LIN {X 0,Y 441.31,Z 713.297,A -85,B 0,C 180,E1 21599.481,E2 21599.481} C_VEL
LIN {X 0,Y 441.247,Z 716.806,A -85,B 0,C 180,E1 21597.403,E2 21597.403} C_VEL
LIN {X 0,Y 441.266,Z 718.402,A -85,B 0,C 180,E1 21595.322,E2 21595.322} C_VEL
LIN {X 0,Y 441.352,Z 718.291,A -85,B 0,C 180,E1 21593.366,E2 21593.366} C_VEL
LIN {X 0,Y 441.5,Z 716.286,A -85,B 0,C 180,E1 21591.273,E2 21591.273} C_VEL
LIN {X 0,Y 441.746,Z 712.662,A -85,B 0,C 180,E1 21589.304,E2 21589.304} C_VEL
LIN {X 0,Y 442.049,Z 707.079,A -85,B 0,C 180,E1 21587.327,E2 21587.327} C_VEL
LIN {X 0,Y 442.464,Z 699.897,A -85,B 0,C 180,E1 21585.474,E2 21585.474} C_VEL
LIN {X 0,Y 442.948,Z 691.121,A -85,B 0,C 180,E1 21583.746,E2 21583.746} C_VEL
LIN {X 0,Y 443.459,Z 681.227,A -85,B 0,C 180,E1 21582.212,E2 21582.212} C_VEL
LIN {X 0,Y 444.021,Z 669.276,A -85,B 0,C 180,E1 21580.738,E2 21580.738} C_VEL
LIN {X 0,Y 444.497,Z 656.854,A -85,B 0,C 180,E1 21579.526,E2 21579.526} C_VEL
LIN {X 0,Y 444.916,Z 642.754,A -85,B 0,C 180,E1 21578.443,E2 21578.443} C_VEL
LIN {X 0,Y 445.197,Z 627.324,A -85,B 0,C 180,E1 21577.555,E2 21577.555} C_VEL
LIN {X 0,Y 445.338,Z 611.674,A -85,B 0,C 180,E1 21576.911,E2 21576.911} C_VEL
LIN {X 0,Y 445.29,Z 594.343,A -85,B 0,C 180,E1 21576.46,E2 21576.46} C_VEL
LIN {X 0,Y 446.556,Z 505.792,A -85,B 0,C 180,E1 21574.804,E2 21574.804} C_VEL
LIN {X 0,Y 447.572,Z 462.908,A -85,B 0,C 180,E1 21573.926,E2 21573.926} C_VEL
LIN {X 0,Y 449.09,Z 454.637,A -85,B 0,C 180,E1 21573.345,E2 21573.345} C_VEL
LIN {X 0,Y 449.865,Z 411.959,A -85,B 0,C 180,E1 21569.922,E2 21569.922} C_VEL
LIN {X 0,Y 450.238,Z 377.811,A -85,B 0,C 180,E1 21567.266,E2 21567.266} C_VEL
LIN {X 0,Y 450.427,Z 358.214,A -85,B 0,C 180,E1 21565.756,E2 21565.756} C_VEL
LIN {X 0,Y 452.726,Z 358.689,A -85,B 0,C 180,E1 21565.418,E2 21565.418} C_VEL
LIN {X 0,Y 455.691,Z 357.568,A -85,B 0,C 180,E1 21565.147,E2 21565.147} C_VEL
LIN {X 0,Y 456.996,Z 357.12,A -85,B 0,C 180,E1 21565.025,E2 21565.025} C_VEL
LIN {X 0,Y 461.236,Z 356.094,A -85,B 0,C 180,E1 21564.597,E2 21564.597} C_VEL
LIN {X 0,Y 470.221,Z 353.87,A -85,B 0,C 180,E1 21563.727,E2 21563.727} C_VEL
LIN {X 0,Y 470.656,Z 372.168,A -85,B 0,C 180,E1 21562.125,E2 21562.125} C_VEL
LIN {X 0,Y 472.911,Z 388.879,A -85,B 0,C 180,E1 21560.508,E2 21560.508} C_VEL
LIN {X 0,Y 476.938,Z 403.833,A -85,B 0,C 180,E1 21558.912,E2 21558.912} C_VEL
LIN {X 0,Y 482.198,Z 416.087,A -85,B 0,C 180,E1 21557.471,E2 21557.471} C_VEL
LIN {X 0,Y 489.251,Z 427.616,A -85,B 0,C 180,E1 21555.986,E2 21555.986} C_VEL
LIN {X 0,Y 498.516,Z 438.468,A -85,B 0,C 180,E1 21554.438,E2 21554.438} C_VEL
LIN {X 0,Y 508.804,Z 447.18,A -85,B 0,C 180,E1 21553.028,E2 21553.028} C_VEL
LIN {X 0,Y 517.76,Z 453.161,A -85,B 0,C 180,E1 21551.96,E2 21551.96} C_VEL
LIN {X 0,Y 501.787,Z 477.95,A -85,B 0,C 180,E1 21551.418,E2 21551.418} C_VEL
LIN {X 0,Y 491.807,Z 495.847,A -85,B 0,C 180,E1 21550.892,E2 21550.892} C_VEL
LIN {X 0,Y 483.679,Z 513.365,A -85,B 0,C 180,E1 21550.241,E2 21550.241} C_VEL
LIN {X 0,Y 476.055,Z 528.839,A -85,B 0,C 180,E1 21549.68,E2 21549.68} C_VEL
LIN {X 0,Y 467.291,Z 551.983,A -85,B 0,C 180,E1 21548.665,E2 21548.665} C_VEL
LIN {X 0,Y 465.606,Z 571.959,A -85,B 0,C 180,E1 21548.437,E2 21548.437} C_VEL
LIN {X 0,Y 464.664,Z 601.449,A -85,B 0,C 180,E1 21547.884,E2 21547.884} C_VEL
LIN {X 0,Y 462.976,Z 626.356,A -85,B 0,C 180,E1 21547.202,E2 21547.202} C_VEL
LIN {X 0,Y 461.15,Z 649.493,A -85,B 0,C 180,E1 21546.332,E2 21546.332} C_VEL
LIN {X 0,Y 459.06,Z 672.171,A -85,B 0,C 180,E1 21545.238,E2 21545.238} C_VEL
LIN {X 0,Y 456.925,Z 693.284,A -85,B 0,C 180,E1 21543.969,E2 21543.969} C_VEL
LIN {X 0,Y 454.675,Z 713.158,A -85,B 0,C 180,E1 21542.525,E2 21542.525} C_VEL
LIN {X 0,Y 452.365,Z 732.465,A -85,B 0,C 180,E1 21540.85,E2 21540.85} C_VEL
LIN {X 0,Y 450.053,Z 750.796,A -85,B 0,C 180,E1 21538.968,E2 21538.968} C_VEL
LIN {X 0,Y 448.043,Z 766.471,A -85,B 0,C 180,E1 21537.076,E2 21537.076} C_VEL
LIN {X 0,Y 445.95,Z 782.819,A -85,B 0,C 180,E1 21534.764,E2 21534.764} C_VEL
LIN {X 0,Y 444.103,Z 797.993,A -85,B 0,C 180,E1 21532.225,E2 21532.225} C_VEL
LIN {X 0,Y 442.674,Z 810.867,A -85,B 0,C 180,E1 21529.667,E2 21529.667} C_VEL
LIN {X 0,Y 441.61,Z 821.723,A -85,B 0,C 180,E1 21527.118,E2 21527.118} C_VEL
LIN {X 0,Y 440.892,Z 830.109,A -85,B 0,C 180,E1 21524.714,E2 21524.714} C_VEL
LIN {X 0,Y 440.36,Z 837.91,A -85,B 0,C 180,E1 21521.924,E2 21521.924} C_VEL
LIN {X 0,Y 440.073,Z 843.957,A -85,B 0,C 180,E1 21519.151,E2 21519.151} C_VEL
LIN {X 0,Y 439.945,Z 848.518,A -85,B 0,C 180,E1 21516.263,E2 21516.263} C_VEL
LIN {X 0,Y 439.913,Z 851.322,A -85,B 0,C 180,E1 21513.388,E2 21513.388} C_VEL
LIN {X 0,Y 439.9,Z 852.433,A -85,B 0,C 180,E1 21510.651,E2 21510.651} C_VEL
LIN {X 0,Y 439.908,Z 852.059,A -85,B 0,C 180,E1 21507.916,E2 21507.916} C_VEL
LIN {X 0,Y 439.928,Z 849.995,A -85,B 0,C 180,E1 21505.045,E2 21505.045} C_VEL
LIN {X 0,Y 439.994,Z 846.441,A -85,B 0,C 180,E1 21502.295,E2 21502.295} C_VEL
LIN {X 0,Y 440.187,Z 841.303,A -85,B 0,C 180,E1 21499.53,E2 21499.53} C_VEL
LIN {X 0,Y 440.603,Z 834.074,A -85,B 0,C 180,E1 21496.616,E2 21496.616} C_VEL
LIN {X 0,Y 441.306,Z 825.238,A -85,B 0,C 180,E1 21493.818,E2 21493.818} C_VEL
LIN {X 0,Y 442.298,Z 814.509,A -85,B 0,C 180,E1 21491.139,E2 21491.139} C_VEL
LIN {X 0,Y 443.609,Z 802.21,A -85,B 0,C 180,E1 21488.57,E2 21488.57} C_VEL
LIN {X 0,Y 445.321,Z 787.723,A -85,B 0,C 180,E1 21486.021,E2 21486.021} C_VEL
LIN {X 0,Y 447.299,Z 772.076,A -85,B 0,C 180,E1 21483.684,E2 21483.684} C_VEL
LIN {X 0,Y 449.449,Z 755.39,A -85,B 0,C 180,E1 21481.571,E2 21481.571} C_VEL
LIN {X 0,Y 451.639,Z 737.833,A -85,B 0,C 180,E1 21479.684,E2 21479.684} C_VEL
LIN {X 0,Y 453.899,Z 719.372,A -85,B 0,C 180,E1 21478.004,E2 21478.004} C_VEL
LIN {X 0,Y 456.25,Z 698.41,A -85,B 0,C 180,E1 21476.403,E2 21476.403} C_VEL
LIN {X 0,Y 458.447,Z 677.594,A -85,B 0,C 180,E1 21475.089,E2 21475.089} C_VEL
LIN {X 0,Y 460.567,Z 654.75,A -85,B 0,C 180,E1 21473.923,E2 21473.923} C_VEL
LIN {X 0,Y 462.537,Z 631.096,A -85,B 0,C 180,E1 21472.979,E2 21472.979} C_VEL
LIN {X 0,Y 464.236,Z 606.974,A -85,B 0,C 180,E1 21472.264,E2 21472.264} C_VEL
LIN {X 0,Y 465.339,Z 581.339,A -85,B 0,C 180,E1 21471.733,E2 21471.733} C_VEL
LIN {X 0,Y 466.057,Z 564.773,A -85,B 0,C 180,E1 21471.482,E2 21471.482} C_VEL
LIN {X 0,Y 467.707,Z 551.654,A -85,B 0,C 180,E1 21471.374,E2 21471.374} C_VEL
LIN {X 0,Y 477.558,Z 530.927,A -85,B 0,C 180,E1 21470.314,E2 21470.314} C_VEL
LIN {X 0,Y 486.134,Z 516.787,A -85,B 0,C 180,E1 21469.734,E2 21469.734} C_VEL
LIN {X 0,Y 489.633,Z 511.052,A -85,B 0,C 180,E1 21469.505,E2 21469.505} C_VEL
LIN {X 0,Y 498.006,Z 497.269,A -85,B 0,C 180,E1 21468.964,E2 21468.964} C_VEL
LIN {X 0,Y 508.107,Z 482.89,A -85,B 0,C 180,E1 21468.507,E2 21468.507} C_VEL
LIN {X 0,Y 496.95,Z 474.729,A -85,B 0,C 180,E1 21467.084,E2 21467.084} C_VEL
LIN {X 0,Y 487.939,Z 465.801,A -85,B 0,C 180,E1 21465.655,E2 21465.655} C_VEL
LIN {X 0,Y 479.934,Z 454.887,A -85,B 0,C 180,E1 21464.048,E2 21464.048} C_VEL
LIN {X 0,Y 473.616,Z 442.126,A -85,B 0,C 180,E1 21462.333,E2 21462.333} C_VEL
LIN {X 0,Y 469.457,Z 428.618,A -85,B 0,C 180,E1 21460.671,E2 21460.671} C_VEL
LIN {X 0,Y 467.031,Z 413.137,A -85,B 0,C 180,E1 21458.928,E2 21458.928} C_VEL
LIN {X 0,Y 466.547,Z 395.635,A -85,B 0,C 180,E1 21457.132,E2 21457.132} C_VEL
LIN {X 0,Y 468.647,Z 371.257,A -85,B 0,C 180,E1 21454.874,E2 21454.874} C_VEL
LIN {X 0,Y 473.371,Z 332.942,A -85,B 0,C 180,E1 21451.354,E2 21451.354} C_VEL
LIN {X 0,Y 474.437,Z 324.206,A -85,B 0,C 180,E1 21450.524,E2 21450.524} C_VEL
LIN {X 0,Y 472.382,Z 319.564,A -85,B 0,C 180,E1 21449.689,E2 21449.689} C_VEL
LIN {X 0,Y 459.708,Z 323.981,A -85,B 0,C 180,E1 21448.251,E2 21448.251} C_VEL
LIN {X 0,Y 456.047,Z 325.473,A -85,B 0,C 180,E1 21447.839,E2 21447.839} C_VEL
LIN {X 0,Y 454.696,Z 325.707,A -85,B 0,C 180,E1 21447.644,E2 21447.644} C_VEL
LIN {X 0,Y 451.321,Z 327.431,A -85,B 0,C 180,E1 21447.296,E2 21447.296} C_VEL
LIN {X 0,Y 449.211,Z 327.424,A -85,B 0,C 180,E1 21446.933,E2 21446.933} C_VEL
LIN {X 0,Y 449.092,Z 328.377,A -85,B 0,C 180,E1 21446.833,E2 21446.833} C_VEL
LIN {X 0,Y 449.024,Z 370.776,A -85,B 0,C 180,E1 21443.838,E2 21443.838} C_VEL
LIN {X 0,Y 448.575,Z 410.447,A -85,B 0,C 180,E1 21440.941,E2 21440.941} C_VEL
LIN {X 0,Y 447.941,Z 450.813,A -85,B 0,C 180,E1 21437.94,E2 21437.94} C_VEL
LIN {X 0,Y 446.95,Z 498.341,A -85,B 0,C 180,E1 21434.311,E2 21434.311} C_VEL
LIN {X 0,Y 446.191,Z 505.272,A -85,B 0,C 180,E1 21433.807,E2 21433.807} C_VEL
LIN {X 0,Y 445.602,Z 509.643,A -85,B 0,C 180,E1 21433.55,E2 21433.55} C_VEL
LIN {X 0,Y 444.21,Z 612.79,A -85,B 0,C 180,E1 21431.634,E2 21431.634} C_VEL
LIN {X 0,Y 444.282,Z 628.686,A -85,B 0,C 180,E1 21431.233,E2 21431.233} C_VEL
LIN {X 0,Y 444.211,Z 642.86,A -85,B 0,C 180,E1 21430.636,E2 21430.636} C_VEL
LIN {X 0,Y 443.957,Z 656.864,A -85,B 0,C 180,E1 21429.79,E2 21429.79} C_VEL
LIN {X 0,Y 443.645,Z 668.929,A -85,B 0,C 180,E1 21428.815,E2 21428.815} C_VEL
LIN {X 0,Y 443.263,Z 680.207,A -85,B 0,C 180,E1 21427.647,E2 21427.647} C_VEL
LIN {X 0,Y 442.814,Z 690.888,A -85,B 0,C 180,E1 21426.222,E2 21426.222} C_VEL
LIN {X 0,Y 442.37,Z 700.16,A -85,B 0,C 180,E1 21424.605,E2 21424.605} C_VEL
LIN {X 0,Y 442.001,Z 707.194,A -85,B 0,C 180,E1 21422.982,E2 21422.982} C_VEL
LIN {X 0,Y 441.71,Z 712.589,A -85,B 0,C 180,E1 21421.297,E2 21421.297} C_VEL
LIN {X 0,Y 441.489,Z 716.487,A -85,B 0,C 180,E1 21419.48,E2 21419.48} C_VEL
LIN {X 0,Y 441.342,Z 718.658,A -85,B 0,C 180,E1 21417.559,E2 21417.559} C_VEL
LIN {X 0,Y 441.266,Z 718.978,A -85,B 0,C 180,E1 21415.711,E2 21415.711} C_VEL
LIN {X 0,Y 441.257,Z 717.447,A -85,B 0,C 180,E1 21413.755,E2 21413.755} C_VEL
LIN {X 0,Y 441.33,Z 713.947,A -85,B 0,C 180,E1 21411.794,E2 21411.794} C_VEL
LIN {X 0,Y 441.485,Z 708.733,A -85,B 0,C 180,E1 21409.957,E2 21409.957} C_VEL
LIN {X 0,Y 441.731,Z 701.958,A -85,B 0,C 180,E1 21408.245,E2 21408.245} C_VEL
LIN {X 0,Y 442.065,Z 693.742,A -85,B 0,C 180,E1 21406.661,E2 21406.661} C_VEL
LIN {X 0,Y 442.465,Z 683.597,A -85,B 0,C 180,E1 21405.138,E2 21405.138} C_VEL
LIN {X 0,Y 442.913,Z 671.646,A -85,B 0,C 180,E1 21403.744,E2 21403.744} C_VEL
LIN {X 0,Y 443.332,Z 658.276,A -85,B 0,C 180,E1 21402.544,E2 21402.544} C_VEL
LIN {X 0,Y 443.71,Z 643.693,A -85,B 0,C 180,E1 21401.567,E2 21401.567} C_VEL
LIN {X 0,Y 443.932,Z 628.136,A -85,B 0,C 180,E1 21400.831,E2 21400.831} C_VEL
LIN {X 0,Y 444.01,Z 611.925,A -85,B 0,C 180,E1 21400.356,E2 21400.356} C_VEL
LIN {X 0,Y 445.329,Z 500.655,A -85,B 0,C 180,E1 21398.361,E2 21398.361} C_VEL
LIN {X 0,Y 446.496,Z 463.1,A -85,B 0,C 180,E1 21395.384,E2 21395.384} C_VEL
LIN {X 0,Y 447.828,Z 415.62,A -85,B 0,C 180,E1 21391.603,E2 21391.603} C_VEL
LIN {X 0,Y 449.089,Z 369.562,A -85,B 0,C 180,E1 21387.926,E2 21387.926} C_VEL
LIN {X 0,Y 450.218,Z 325.21,A -85,B 0,C 180,E1 21384.374,E2 21384.374} C_VEL
LIN {X 0,Y 451.153,Z 287.779,A -85,B 0,C 180,E1 21381.373,E2 21381.373} C_VEL
LIN {X 0,Y 449.471,Z 282.336,A -85,B 0,C 180,E1 21380.798,E2 21380.798} C_VEL
LIN {X 0,Y 451.314,Z 282.535,A -85,B 0,C 180,E1 21380.353,E2 21380.353} C_VEL
LIN {X 0,Y 453.906,Z 282.47,A -85,B 0,C 180,E1 21379.802,E2 21379.802} C_VEL
LIN {X 0,Y 458.201,Z 291.634,A -85,B 0,C 180,E1 21377.431,E2 21377.431} C_VEL
LIN {X 0,Y 463.301,Z 302.907,A -85,B 0,C 180,E1 21374.763,E2 21374.763} C_VEL
LIN {X 0,Y 468.848,Z 316.513,A -85,B 0,C 180,E1 21371.902,E2 21371.902} C_VEL
LIN {X 0,Y 467.094,Z 330.439,A -85,B 0,C 180,E1 21370.366,E2 21370.366} C_VEL
LIN {X 0,Y 467.778,Z 334.267,A -85,B 0,C 180,E1 21370.217,E2 21370.217} C_VEL
LIN {X 0,Y 467.35,Z 351.287,A -85,B 0,C 180,E1 21369.928,E2 21369.928} C_VEL
LIN {X 0,Y 466.406,Z 358.984,A -85,B 0,C 180,E1 21369.877,E2 21369.877} C_VEL
LIN {X 0,Y 461.125,Z 379.53,A -85,B 0,C 180,E1 21370.025,E2 21370.025} C_VEL
LIN {X 0,Y 460.345,Z 386.128,A -85,B 0,C 180,E1 21369.967,E2 21369.967} C_VEL
LIN {X 0,Y 457.193,Z 465.291,A -85,B 0,C 180,E1 21368.444,E2 21368.444} C_VEL
LIN {X 0,Y 452.322,Z 565.562,A -85,B 0,C 180,E1 21366.246,E2 21366.246} C_VEL
LIN {X 0,Y 451.213,Z 587.266,A -85,B 0,C 180,E1 21365.631,E2 21365.631} C_VEL
LIN {X 0,Y 449.865,Z 607.038,A -85,B 0,C 180,E1 21364.835,E2 21364.835} C_VEL
LIN {X 0,Y 448.196,Z 626.387,A -85,B 0,C 180,E1 21363.821,E2 21363.821} C_VEL
LIN {X 0,Y 446.216,Z 645.87,A -85,B 0,C 180,E1 21362.533,E2 21362.533} C_VEL
LIN {X 0,Y 444.104,Z 664.276,A -85,B 0,C 180,E1 21361.036,E2 21361.036} C_VEL
LIN {X 0,Y 441.961,Z 681.656,A -85,B 0,C 180,E1 21359.327,E2 21359.327} C_VEL
LIN {X 0,Y 439.837,Z 698.057,A -85,B 0,C 180,E1 21357.396,E2 21357.396} C_VEL
LIN {X 0,Y 437.884,Z 713.133,A -85,B 0,C 180,E1 21355.277,E2 21355.277} C_VEL
LIN {X 0,Y 436.225,Z 726.308,A -85,B 0,C 180,E1 21353.076,E2 21353.076} C_VEL
LIN {X 0,Y 434.786,Z 738.681,A -85,B 0,C 180,E1 21350.601,E2 21350.601} C_VEL
LIN {X 0,Y 433.68,Z 749.378,A -85,B 0,C 180,E1 21347.996,E2 21347.996} C_VEL
LIN {X 0,Y 432.923,Z 757.949,A -85,B 0,C 180,E1 21345.403,E2 21345.403} C_VEL
LIN {X 0,Y 432.469,Z 764.659,A -85,B 0,C 180,E1 21342.824,E2 21342.824} C_VEL
LIN {X 0,Y 432.223,Z 769.704,A -85,B 0,C 180,E1 21340.261,E2 21340.261} C_VEL
LIN {X 0,Y 432.09,Z 773.262,A -85,B 0,C 180,E1 21337.579,E2 21337.579} C_VEL
LIN {X 0,Y 432.051,Z 775.178,A -85,B 0,C 180,E1 21334.912,E2 21334.912} C_VEL
LIN {X 0,Y 432.036,Z 775.537,A -85,B 0,C 180,E1 21332.255,E2 21332.255} C_VEL
LIN {X 0,Y 432.061,Z 774.353,A -85,B 0,C 180,E1 21329.602,E2 21329.602} C_VEL
LIN {X 0,Y 432.141,Z 771.617,A -85,B 0,C 180,E1 21326.95,E2 21326.95} C_VEL
LIN {X 0,Y 432.331,Z 767.214,A -85,B 0,C 180,E1 21324.293,E2 21324.293} C_VEL
LIN {X 0,Y 432.692,Z 761.063,A -85,B 0,C 180,E1 21321.629,E2 21321.629} C_VEL
LIN {X 0,Y 433.289,Z 753.478,A -85,B 0,C 180,E1 21319.092,E2 21319.092} C_VEL
LIN {X 0,Y 434.198,Z 744.012,A -85,B 0,C 180,E1 21316.551,E2 21316.551} C_VEL
LIN {X 0,Y 435.402,Z 733.057,A -85,B 0,C 180,E1 21314.141,E2 21314.141} C_VEL
LIN {X 0,Y 436.888,Z 720.66,A -85,B 0,C 180,E1 21311.865,E2 21311.865} C_VEL
LIN {X 0,Y 438.636,Z 706.804,A -85,B 0,C 180,E1 21309.728,E2 21309.728} C_VEL
LIN {X 0,Y 440.487,Z 692.349,A -85,B 0,C 180,E1 21307.839,E2 21307.839} C_VEL
LIN {X 0,Y 442.487,Z 676.355,A -85,B 0,C 180,E1 21306.071,E2 21306.071} C_VEL
LIN {X 0,Y 444.607,Z 658.422,A -85,B 0,C 180,E1 21304.419,E2 21304.419} C_VEL
LIN {X 0,Y 446.669,Z 639.282,A -85,B 0,C 180,E1 21302.973,E2 21302.973} C_VEL
LIN {X 0,Y 448.497,Z 619.99,A -85,B 0,C 180,E1 21301.795,E2 21301.795} C_VEL
LIN {X 0,Y 450.083,Z 599.348,A -85,B 0,C 180,E1 21300.811,E2 21300.811} C_VEL
LIN {X 0,Y 451.333,Z 578.519,A -85,B 0,C 180,E1 21300.079,E2 21300.079} C_VEL
LIN {X 0,Y 453.796,Z 525.708,A -85,B 0,C 180,E1 21298.853,E2 21298.853} C_VEL
LIN {X 0,Y 457.817,Z 435.454,A -85,B 0,C 180,E1 21296.979,E2 21296.979} C_VEL
LIN {X 0,Y 460.313,Z 359.092,A -85,B 0,C 180,E1 21295.584,E2 21295.584} C_VEL
LIN {X 0,Y 460.863,Z 329.957,A -85,B 0,C 180,E1 21295.07,E2 21295.07} C_VEL
LIN {X 0,Y 462.111,Z 317.947,A -85,B 0,C 180,E1 21293.948,E2 21293.948} C_VEL
LIN {X 0,Y 454.634,Z 301.125,A -85,B 0,C 180,E1 21290.928,E2 21290.928} C_VEL
LIN {X 0,Y 447.804,Z 286.639,A -85,B 0,C 180,E1 21288.033,E2 21288.033} C_VEL
LIN {X 0,Y 442.473,Z 276.494,A -85,B 0,C 180,E1 21285.753,E2 21285.753} C_VEL
LIN {X 0,Y 440.585,Z 272.815,A -85,B 0,C 180,E1 21284.893,E2 21284.893} C_VEL
LIN {X 0,Y 438.087,Z 268.159,A -85,B 0,C 180,E1 21283.753,E2 21283.753} C_VEL
LIN {X 0,Y 436.13,Z 264.36,A -85,B 0,C 180,E1 21282.809,E2 21282.809} C_VEL
LIN {X 0,Y 433.527,Z 260.102,A -85,B 0,C 180,E1 21281.624,E2 21281.624} C_VEL
LIN {X 0,Y 433.246,Z 258.749,A -85,B 0,C 180,E1 21281.304,E2 21281.304} C_VEL
LIN {X 0,Y 433.251,Z 258.747,A -85,B 0,C 180,E1 21277.37,E2 21277.37} C_VEL
LIN {X 0,Y 433.293,Z 258.995,A -85,B 0,C 180,E1 21273.948,E2 21273.948} C_VEL
LIN {X 0,Y 442.041,Z 284.911,A -85,B 0,C 180,E1 21270.988,E2 21270.988} C_VEL
LIN {X 0,Y 444.141,Z 292.371,A -85,B 0,C 180,E1 21270.177,E2 21270.177} C_VEL
LIN {X 0,Y 443.072,Z 334.296,A -85,B 0,C 180,E1 21266.54,E2 21266.54} C_VEL
LIN {X 0,Y 441.851,Z 375.973,A -85,B 0,C 180,E1 21262.927,E2 21262.927} C_VEL
LIN {X 0,Y 440.518,Z 419.079,A -85,B 0,C 180,E1 21259.215,E2 21259.215} C_VEL
LIN {X 0,Y 439.579,Z 452.59,A -85,B 0,C 180,E1 21256.369,E2 21256.369} C_VEL
LIN {X 0,Y 437.55,Z 596.495,A -85,B 0,C 180,E1 21253.669,E2 21253.669} C_VEL
LIN {X 0,Y 437.364,Z 613.001,A -85,B 0,C 180,E1 21253.123,E2 21253.123} C_VEL
LIN {X 0,Y 436.985,Z 628.731,A -85,B 0,C 180,E1 21252.354,E2 21252.354} C_VEL
LIN {X 0,Y 436.5,Z 643.911,A -85,B 0,C 180,E1 21251.362,E2 21251.362} C_VEL
LIN {X 0,Y 435.911,Z 658.647,A -85,B 0,C 180,E1 21250.107,E2 21250.107} C_VEL
LIN {X 0,Y 435.319,Z 671.504,A -85,B 0,C 180,E1 21248.72,E2 21248.72} C_VEL
LIN {X 0,Y 434.748,Z 683.332,A -85,B 0,C 180,E1 21247.135,E2 21247.135} C_VEL
LIN {X 0,Y 434.242,Z 693.486,A -85,B 0,C 180,E1 21245.418,E2 21245.418} C_VEL
LIN {X 0,Y 433.861,Z 702.174,A -85,B 0,C 180,E1 21243.568,E2 21243.568} C_VEL
LIN {X 0,Y 433.586,Z 709.271,A -85,B 0,C 180,E1 21241.586,E2 21241.586} C_VEL
LIN {X 0,Y 433.428,Z 714.441,A -85,B 0,C 180,E1 21239.604,E2 21239.604} C_VEL
LIN {X 0,Y 433.362,Z 718.07,A -85,B 0,C 180,E1 21237.478,E2 21237.478} C_VEL
LIN {X 0,Y 433.385,Z 719.768,A -85,B 0,C 180,E1 21235.369,E2 21235.369} C_VEL
LIN {X 0,Y 433.488,Z 719.674,A -85,B 0,C 180,E1 21233.245,E2 21233.245} C_VEL
LIN {X 0,Y 433.663,Z 717.629,A -85,B 0,C 180,E1 21231.114,E2 21231.114} C_VEL
LIN {X 0,Y 433.935,Z 713.935,A -85,B 0,C 180,E1 21229.109,E2 21229.109} C_VEL
LIN {X 0,Y 434.279,Z 708.27,A -85,B 0,C 180,E1 21227.096,E2 21227.096} C_VEL
LIN {X 0,Y 434.697,Z 701.549,A -85,B 0,C 180,E1 21225.345,E2 21225.345} C_VEL
LIN {X 0,Y 435.219,Z 692.807,A -85,B 0,C 180,E1 21223.586,E2 21223.586} C_VEL
LIN {X 0,Y 435.775,Z 682.834,A -85,B 0,C 180,E1 21222.009,E2 21222.009} C_VEL
LIN {X 0,Y 436.363,Z 670.994,A -85,B 0,C 180,E1 21220.526,E2 21220.526} C_VEL
LIN {X 0,Y 436.863,Z 658.545,A -85,B 0,C 180,E1 21219.292,E2 21219.292} C_VEL
LIN {X 0,Y 437.318,Z 644.116,A -85,B 0,C 180,E1 21218.166,E2 21218.166} C_VEL
LIN {X 0,Y 437.618,Z 628.458,A -85,B 0,C 180,E1 21217.254,E2 21217.254} C_VEL
LIN {X 0,Y 437.758,Z 612.739,A -85,B 0,C 180,E1 21216.603,E2 21216.603} C_VEL
LIN {X 0,Y 437.7,Z 595.749,A -85,B 0,C 180,E1 21216.158,E2 21216.158} C_VEL
LIN {X 0,Y 439.034,Z 510.998,A -85,B 0,C 180,E1 21214.517,E2 21214.517} C_VEL
LIN {X 0,Y 440.259,Z 464.842,A -85,B 0,C 180,E1 21213.533,E2 21213.533} C_VEL
LIN {X 0,Y 441.927,Z 455.489,A -85,B 0,C 180,E1 21212.878,E2 21212.878} C_VEL
LIN {X 0,Y 442.765,Z 415.162,A -85,B 0,C 180,E1 21209.613,E2 21209.613} C_VEL
LIN {X 0,Y 443.239,Z 379.479,A -85,B 0,C 180,E1 21206.815,E2 21206.815} C_VEL
LIN {X 0,Y 443.412,Z 367.038,A -85,B 0,C 180,E1 21205.843,E2 21205.843} C_VEL
LIN {X 0,Y 445.366,Z 367.478,A -85,B 0,C 180,E1 21205.546,E2 21205.546} C_VEL
LIN {X 0,Y 447.835,Z 366.737,A -85,B 0,C 180,E1 21205.297,E2 21205.297} C_VEL
LIN {X 0,Y 449.66,Z 365.839,A -85,B 0,C 180,E1 21205.148,E2 21205.148} C_VEL
LIN {X 0,Y 453.63,Z 365.011,A -85,B 0,C 180,E1 21204.727,E2 21204.727} C_VEL
LIN {X 0,Y 456.213,Z 364.067,A -85,B 0,C 180,E1 21204.495,E2 21204.495} C_VEL
LIN {X 0,Y 463.812,Z 362.167,A -85,B 0,C 180,E1 21203.754,E2 21203.754} C_VEL
LIN {X 0,Y 464.754,Z 381.015,A -85,B 0,C 180,E1 21202.027,E2 21202.027} C_VEL
LIN {X 0,Y 467.442,Z 397.094,A -85,B 0,C 180,E1 21200.401,E2 21200.401} C_VEL
LIN {X 0,Y 471.69,Z 411.162,A -85,B 0,C 180,E1 21198.839,E2 21198.839} C_VEL
LIN {X 0,Y 478.084,Z 424.746,A -85,B 0,C 180,E1 21197.18,E2 21197.18} C_VEL
LIN {X 0,Y 485.424,Z 435.689,A -85,B 0,C 180,E1 21195.713,E2 21195.713} C_VEL
LIN {X 0,Y 494.918,Z 446.101,A -85,B 0,C 180,E1 21194.178,E2 21194.178} C_VEL
LIN {X 0,Y 506.052,Z 454.995,A -85,B 0,C 180,E1 21192.693,E2 21192.693} C_VEL
LIN {X 0,Y 508.227,Z 456.583,A -85,B 0,C 180,E1 21192.421,E2 21192.421} C_VEL
LIN {X 0,Y 493.974,Z 479.096,A -85,B 0,C 180,E1 21191.91,E2 21191.91} C_VEL
LIN {X 0,Y 484.208,Z 497.036,A -85,B 0,C 180,E1 21191.36,E2 21191.36} C_VEL
LIN {X 0,Y 477.395,Z 511.775,A -85,B 0,C 180,E1 21190.803,E2 21190.803} C_VEL
LIN {X 0,Y 469.738,Z 527.205,A -85,B 0,C 180,E1 21190.242,E2 21190.242} C_VEL
LIN {X 0,Y 461.072,Z 549.727,A -85,B 0,C 180,E1 21189.257,E2 21189.257} C_VEL
LIN {X 0,Y 459.096,Z 571.202,A -85,B 0,C 180,E1 21189.024,E2 21189.024} C_VEL
LIN {X 0,Y 458.106,Z 599.923,A -85,B 0,C 180,E1 21188.476,E2 21188.476} C_VEL
LIN {X 0,Y 456.306,Z 625.104,A -85,B 0,C 180,E1 21187.781,E2 21187.781} C_VEL
LIN {X 0,Y 454.415,Z 648.011,A -85,B 0,C 180,E1 21186.919,E2 21186.919} C_VEL
LIN {X 0,Y 452.238,Z 670.792,A -85,B 0,C 180,E1 21185.823,E2 21185.823} C_VEL
LIN {X 0,Y 449.943,Z 692.453,A -85,B 0,C 180,E1 21184.518,E2 21184.518} C_VEL
LIN {X 0,Y 447.674,Z 711.668,A -85,B 0,C 180,E1 21183.119,E2 21183.119} C_VEL
LIN {X 0,Y 445.379,Z 730.006,A -85,B 0,C 180,E1 21181.539,E2 21181.539} C_VEL
LIN {X 0,Y 443.087,Z 747.448,A -85,B 0,C 180,E1 21179.765,E2 21179.765} C_VEL
LIN {X 0,Y 440.843,Z 763.889,A -85,B 0,C 180,E1 21177.805,E2 21177.805} C_VEL
LIN {X 0,Y 438.504,Z 781.042,A -85,B 0,C 180,E1 21175.383,E2 21175.383} C_VEL
LIN {X 0,Y 436.575,Z 795.731,A -85,B 0,C 180,E1 21172.914,E2 21172.914} C_VEL
LIN {X 0,Y 435.07,Z 808.246,A -85,B 0,C 180,E1 21170.446,E2 21170.446} C_VEL
LIN {X 0,Y 433.826,Z 819.974,A -85,B 0,C 180,E1 21167.712,E2 21167.712} C_VEL
LIN {X 0,Y 432.894,Z 830.504,A -85,B 0,C 180,E1 21164.718,E2 21164.718} C_VEL
LIN {X 0,Y 432.344,Z 838.833,A -85,B 0,C 180,E1 21161.743,E2 21161.743} C_VEL
LIN {X 0,Y 432.066,Z 844.434,A -85,B 0,C 180,E1 21159.054,E2 21159.054} C_VEL
LIN {X 0,Y 431.946,Z 848.676,A -85,B 0,C 180,E1 21156.246,E2 21156.246} C_VEL
LIN {X 0,Y 431.914,Z 851.418,A -85,B 0,C 180,E1 21153.318,E2 21153.318} C_VEL
LIN {X 0,Y 431.898,Z 852.447,A -85,B 0,C 180,E1 21150.531,E2 21150.531} C_VEL
LIN {X 0,Y 431.909,Z 851.994,A -85,B 0,C 180,E1 21147.744,E2 21147.744} C_VEL
LIN {X 0,Y 431.931,Z 849.869,A -85,B 0,C 180,E1 21144.82,E2 21144.82} C_VEL
LIN {X 0,Y 432.023,Z 846.023,A -85,B 0,C 180,E1 21141.884,E2 21141.884} C_VEL
LIN {X 0,Y 432.241,Z 840.701,A -85,B 0,C 180,E1 21139.066,E2 21139.066} C_VEL
LIN {X 0,Y 432.654,Z 833.768,A -85,B 0,C 180,E1 21136.366,E2 21136.366} C_VEL
LIN {X 0,Y 433.401,Z 824.533,A -85,B 0,C 180,E1 21133.515,E2 21133.515} C_VEL
LIN {X 0,Y 434.462,Z 813.757,A -85,B 0,C 180,E1 21130.786,E2 21130.786} C_VEL
LIN {X 0,Y 435.851,Z 801.511,A -85,B 0,C 180,E1 21128.183,E2 21128.183} C_VEL
LIN {X 0,Y 437.701,Z 786.979,A -85,B 0,C 180,E1 21125.577,E2 21125.577} C_VEL
LIN {X 0,Y 439.76,Z 771.554,A -85,B 0,C 180,E1 21123.244,E2 21123.244} C_VEL
LIN {X 0,Y 442.064,Z 754.741,A -85,B 0,C 180,E1 21121.081,E2 21121.081} C_VEL
LIN {X 0,Y 444.355,Z 737.56,A -85,B 0,C 180,E1 21119.209,E2 21119.209} C_VEL
LIN {X 0,Y 446.776,Z 718.364,A -85,B 0,C 180,E1 21117.457,E2 21117.457} C_VEL
LIN {X 0,Y 449.204,Z 697.891,A -85,B 0,C 180,E1 21115.881,E2 21115.881} C_VEL
LIN {X 0,Y 451.532,Z 676.814,A -85,B 0,C 180,E1 21114.537,E2 21114.537} C_VEL
LIN {X 0,Y 453.757,Z 654.206,A -85,B 0,C 180,E1 21113.373,E2 21113.373} C_VEL
LIN {X 0,Y 455.871,Z 630.161,A -85,B 0,C 180,E1 21112.402,E2 21112.402} C_VEL
LIN {X 0,Y 457.758,Z 605.242,A -85,B 0,C 180,E1 21111.655,E2 21111.655} C_VEL
LIN {X 0,Y 458.927,Z 579.148,A -85,B 0,C 180,E1 21111.107,E2 21111.107} C_VEL
LIN {X 0,Y 459.698,Z 564.113,A -85,B 0,C 180,E1 21110.885,E2 21110.885} C_VEL
LIN {X 0,Y 461.647,Z 549.225,A -85,B 0,C 180,E1 21110.77,E2 21110.77} C_VEL
LIN {X 0,Y 471.404,Z 529.019,A -85,B 0,C 180,E1 21109.74,E2 21109.74} C_VEL
LIN {X 0,Y 480.085,Z 514.758,A -85,B 0,C 180,E1 21109.159,E2 21109.159} C_VEL
LIN {X 0,Y 483.818,Z 508.625,A -85,B 0,C 180,E1 21108.914,E2 21108.914} C_VEL
LIN {X 0,Y 492.788,Z 494.086,A -85,B 0,C 180,E1 21108.356,E2 21108.356} C_VEL
LIN {X 0,Y 498.44,Z 485.91,A -85,B 0,C 180,E1 21108.091,E2 21108.091} C_VEL
LIN {X 0,Y 487.48,Z 476.951,A -85,B 0,C 180,E1 21106.558,E2 21106.558} C_VEL
LIN {X 0,Y 478.37,Z 466.655,A -85,B 0,C 180,E1 21104.948,E2 21104.948} C_VEL
LIN {X 0,Y 471.506,Z 455.938,A -85,B 0,C 180,E1 21103.398,E2 21103.398} C_VEL
LIN {X 0,Y 465.86,Z 443.033,A -85,B 0,C 180,E1 21101.677,E2 21101.677} C_VEL
LIN {X 0,Y 462.2,Z 429.141,A -85,B 0,C 180,E1 21099.977,E2 21099.977} C_VEL
LIN {X 0,Y 460.208,Z 412.772,A -85,B 0,C 180,E1 21098.141,E2 21098.141} C_VEL
LIN {X 0,Y 460.263,Z 394.702,A -85,B 0,C 180,E1 21096.297,E2 21096.297} C_VEL
LIN {X 0,Y 466.99,Z 338.383,A -85,B 0,C 180,E1 21091.064,E2 21091.064} C_VEL
LIN {X 0,Y 468.301,Z 328.457,A -85,B 0,C 180,E1 21090.115,E2 21090.115} C_VEL
LIN {X 0,Y 467.675,Z 327.214,A -85,B 0,C 180,E1 21089.877,E2 21089.877} C_VEL
LIN {X 0,Y 457.1,Z 331.018,A -85,B 0,C 180,E1 21088.699,E2 21088.699} C_VEL
LIN {X 0,Y 452.525,Z 332.678,A -85,B 0,C 180,E1 21088.164,E2 21088.164} C_VEL
LIN {X 0,Y 448.867,Z 334.182,A -85,B 0,C 180,E1 21087.745,E2 21087.745} C_VEL
LIN {X 0,Y 447.475,Z 334.493,A -85,B 0,C 180,E1 21087.55,E2 21087.55} C_VEL
LIN {X 0,Y 444.83,Z 335.997,A -85,B 0,C 180,E1 21087.292,E2 21087.292} C_VEL
LIN {X 0,Y 442.785,Z 336.42,A -85,B 0,C 180,E1 21086.992,E2 21086.992} C_VEL
LIN {X 0,Y 441.969,Z 336.331,A -85,B 0,C 180,E1 21086.81,E2 21086.81} C_VEL
LIN {X 0,Y 441.726,Z 379.896,A -85,B 0,C 180,E1 21083.689,E2 21083.689} C_VEL
LIN {X 0,Y 441.061,Z 428.671,A -85,B 0,C 180,E1 21080.086,E2 21080.086} C_VEL
LIN {X 0,Y 440.09,Z 475.155,A -85,B 0,C 180,E1 21076.559,E2 21076.559} C_VEL
LIN {X 0,Y 439.366,Z 502.764,A -85,B 0,C 180,E1 21074.429,E2 21074.429} C_VEL
LIN {X 0,Y 438.069,Z 511.202,A -85,B 0,C 180,E1 21073.88,E2 21073.88} C_VEL
LIN {X 0,Y 436.526,Z 613.091,A -85,B 0,C 180,E1 21071.921,E2 21071.921} C_VEL
LIN {X 0,Y 436.619,Z 629.794,A -85,B 0,C 180,E1 21071.504,E2 21071.504} C_VEL
LIN {X 0,Y 436.548,Z 644.174,A -85,B 0,C 180,E1 21070.891,E2 21070.891} C_VEL
LIN {X 0,Y 436.304,Z 657.311,A -85,B 0,C 180,E1 21070.096,E2 21070.096} C_VEL
LIN {X 0,Y 435.978,Z 669.652,A -85,B 0,C 180,E1 21069.104,E2 21069.104} C_VEL
LIN {X 0,Y 435.544,Z 681.641,A -85,B 0,C 180,E1 21067.85,E2 21067.85} C_VEL
LIN {X 0,Y 435.08,Z 691.88,A -85,B 0,C 180,E1 21066.465,E2 21066.465} C_VEL
LIN {X 0,Y 434.616,Z 700.955,A -85,B 0,C 180,E1 21064.882,E2 21064.882} C_VEL
LIN {X 0,Y 434.23,Z 707.915,A -85,B 0,C 180,E1 21063.3,E2 21063.3} C_VEL
LIN {X 0,Y 433.883,Z 713.867,A -85,B 0,C 180,E1 21061.452,E2 21061.452} C_VEL
LIN {X 0,Y 433.623,Z 718.018,A -85,B 0,C 180,E1 21059.471,E2 21059.471} C_VEL
LIN {X 0,Y 433.459,Z 720.102,A -85,B 0,C 180,E1 21057.488,E2 21057.488} C_VEL
LIN {X 0,Y 433.377,Z 720.281,A -85,B 0,C 180,E1 21055.633,E2 21055.633} C_VEL
LIN {X 0,Y 433.365,Z 718.802,A -85,B 0,C 180,E1 21053.774,E2 21053.774} C_VEL
LIN {X 0,Y 433.438,Z 715.294,A -85,B 0,C 180,E1 21051.777,E2 21051.777} C_VEL
LIN {X 0,Y 433.601,Z 710.059,A -85,B 0,C 180,E1 21049.906,E2 21049.906} C_VEL
LIN {X 0,Y 433.857,Z 703.26,A -85,B 0,C 180,E1 21048.164,E2 21048.164} C_VEL
LIN {X 0,Y 434.207,Z 695.019,A -85,B 0,C 180,E1 21046.551,E2 21046.551} C_VEL
LIN {X 0,Y 434.626,Z 684.844,A -85,B 0,C 180,E1 21045,E2 21045} C_VEL
LIN {X 0,Y 435.095,Z 672.852,A -85,B 0,C 180,E1 21043.581,E2 21043.581} C_VEL
LIN {X 0,Y 435.532,Z 659.437,A -85,B 0,C 180,E1 21042.359,E2 21042.359} C_VEL
LIN {X 0,Y 435.921,Z 644.906,A -85,B 0,C 180,E1 21041.37,E2 21041.37} C_VEL
LIN {X 0,Y 436.153,Z 629.19,A -85,B 0,C 180,E1 21040.615,E2 21040.615} C_VEL
LIN {X 0,Y 436.231,Z 612.982,A -85,B 0,C 180,E1 21040.133,E2 21040.133} C_VEL
LIN {X 0,Y 437.612,Z 501.821,A -85,B 0,C 180,E1 21038.099,E2 21038.099} C_VEL
LIN {X 0,Y 438.602,Z 474.464,A -85,B 0,C 180,E1 21035.917,E2 21035.917} C_VEL
LIN {X 0,Y 439.975,Z 426.686,A -85,B 0,C 180,E1 21032.086,E2 21032.086} C_VEL
LIN {X 0,Y 441.329,Z 380.978,A -85,B 0,C 180,E1 21028.415,E2 21028.415} C_VEL
LIN {X 0,Y 442.52,Z 337.715,A -85,B 0,C 180,E1 21024.925,E2 21024.925} C_VEL
LIN {X 0,Y 443.756,Z 290.218,A -85,B 0,C 180,E1 21021.096,E2 21021.096} C_VEL
LIN {X 0,Y 443.429,Z 289.131,A -85,B 0,C 180,E1 21020.974,E2 21020.974} C_VEL
LIN {X 0,Y 445.175,Z 289.386,A -85,B 0,C 180,E1 21020.534,E2 21020.534} C_VEL
LIN {X 0,Y 448.886,Z 289.096,A -85,B 0,C 180,E1 21019.762,E2 21019.762} C_VEL
LIN {X 0,Y 454.001,Z 299.891,A -85,B 0,C 180,E1 21016.943,E2 21016.943} C_VEL
LIN {X 0,Y 459.579,Z 312.989,A -85,B 0,C 180,E1 21013.935,E2 21013.935} C_VEL
LIN {X 0,Y 462.684,Z 320.953,A -85,B 0,C 180,E1 21012.28,E2 21012.28} C_VEL
LIN {X 0,Y 461.11,Z 332.679,A -85,B 0,C 180,E1 21010.974,E2 21010.974} C_VEL
LIN {X 0,Y 461.703,Z 336.187,A -85,B 0,C 180,E1 21010.837,E2 21010.837} C_VEL
LIN {X 0,Y 460.345,Z 386.128,A -85,B 0,C 180,E1 21009.967,E2 21009.967} C_VEL
LIN {X 0,Y 459.331,Z 393.812,A -85,B 0,C 180,E1 21009.909,E2 21009.909} C_VEL
LIN {X 0,Y 453.843,Z 414.314,A -85,B 0,C 180,E1 21010.043,E2 21010.043} C_VEL
LIN {X 0,Y 452.998,Z 420.902,A -85,B 0,C 180,E1 21009.979,E2 21009.979} C_VEL
LIN {X 0,Y 449.136,Z 502.676,A -85,B 0,C 180,E1 21008.28,E2 21008.28} C_VEL
LIN {X 0,Y 445.17,Z 577.311,A -85,B 0,C 180,E1 21006.527,E2 21006.527} C_VEL
LIN {X 0,Y 443.906,Z 597.827,A -85,B 0,C 180,E1 21005.818,E2 21005.818} C_VEL
LIN {X 0,Y 442.273,Z 617.697,A -85,B 0,C 180,E1 21004.888,E2 21004.888} C_VEL
LIN {X 0,Y 440.347,Z 637.094,A -85,B 0,C 180,E1 21003.723,E2 21003.723} C_VEL
LIN {X 0,Y 438.107,Z 656.381,A -85,B 0,C 180,E1 21002.279,E2 21002.279} C_VEL
LIN {X 0,Y 435.818,Z 674.514,A -85,B 0,C 180,E1 21000.619,E2 21000.619} C_VEL
LIN {X 0,Y 433.575,Z 691.05,A -85,B 0,C 180,E1 20998.798,E2 20998.798} C_VEL
LIN {X 0,Y 431.375,Z 706.843,A -85,B 0,C 180,E1 20996.722,E2 20996.722} C_VEL
LIN {X 0,Y 429.416,Z 721.094,A -85,B 0,C 180,E1 20994.485,E2 20994.485} C_VEL
LIN {X 0,Y 427.749,Z 733.779,A -85,B 0,C 180,E1 20992.107,E2 20992.107} C_VEL
LIN {X 0,Y 426.414,Z 744.932,A -85,B 0,C 180,E1 20989.591,E2 20989.591} C_VEL
LIN {X 0,Y 425.412,Z 754.53,A -85,B 0,C 180,E1 20986.943,E2 20986.943} C_VEL
LIN {X 0,Y 424.762,Z 762.167,A -85,B 0,C 180,E1 20984.31,E2 20984.31} C_VEL
LIN {X 0,Y 424.386,Z 768.059,A -85,B 0,C 180,E1 20981.69,E2 20981.69} C_VEL
LIN {X 0,Y 424.19,Z 772.494,A -85,B 0,C 180,E1 20978.95,E2 20978.95} C_VEL
LIN {X 0,Y 424.099,Z 775.187,A -85,B 0,C 180,E1 20976.226,E2 20976.226} C_VEL
LIN {X 0,Y 424.073,Z 776.279,A -85,B 0,C 180,E1 20973.515,E2 20973.515} C_VEL
LIN {X 0,Y 424.075,Z 775.81,A -85,B 0,C 180,E1 20970.811,E2 20970.811} C_VEL
LIN {X 0,Y 424.133,Z 773.782,A -85,B 0,C 180,E1 20968.109,E2 20968.109} C_VEL
LIN {X 0,Y 424.277,Z 770.162,A -85,B 0,C 180,E1 20965.404,E2 20965.404} C_VEL
LIN {X 0,Y 424.58,Z 764.819,A -85,B 0,C 180,E1 20962.694,E2 20962.694} C_VEL
LIN {X 0,Y 425.079,Z 758.035,A -85,B 0,C 180,E1 20960.113,E2 20960.113} C_VEL
LIN {X 0,Y 425.903,Z 749.481,A -85,B 0,C 180,E1 20957.527,E2 20957.527} C_VEL
LIN {X 0,Y 427,Z 739.538,A -85,B 0,C 180,E1 20955.074,E2 20955.074} C_VEL
LIN {X 0,Y 428.485,Z 727.535,A -85,B 0,C 180,E1 20952.621,E2 20952.621} C_VEL
LIN {X 0,Y 430.278,Z 713.952,A -85,B 0,C 180,E1 20950.309,E2 20950.309} C_VEL
LIN {X 0,Y 432.339,Z 698.713,A -85,B 0,C 180,E1 20948.14,E2 20948.14} C_VEL
LIN {X 0,Y 434.569,Z 682.123,A -85,B 0,C 180,E1 20946.167,E2 20946.167} C_VEL
LIN {X 0,Y 436.802,Z 664.584,A -85,B 0,C 180,E1 20944.431,E2 20944.431} C_VEL
LIN {X 0,Y 438.999,Z 645.849,A -85,B 0,C 180,E1 20942.902,E2 20942.902} C_VEL
LIN {X 0,Y 440.986,Z 626.705,A -85,B 0,C 180,E1 20941.633,E2 20941.633} C_VEL
LIN {X 0,Y 442.708,Z 606.961,A -85,B 0,C 180,E1 20940.594,E2 20940.594} C_VEL
LIN {X 0,Y 444.133,Z 586.198,A -85,B 0,C 180,E1 20939.768,E2 20939.768} C_VEL
LIN {X 0,Y 445.366,Z 561.556,A -85,B 0,C 180,E1 20939.09,E2 20939.09} C_VEL
LIN {X 0,Y 450.11,Z 467.065,A -85,B 0,C 180,E1 20936.994,E2 20936.994} C_VEL
LIN {X 0,Y 453.231,Z 389.759,A -85,B 0,C 180,E1 20935.488,E2 20935.488} C_VEL
LIN {X 0,Y 454.796,Z 332.13,A -85,B 0,C 180,E1 20934.473,E2 20934.473} C_VEL
LIN {X 0,Y 455.943,Z 322.16,A -85,B 0,C 180,E1 20933.538,E2 20933.538} C_VEL
LIN {X 0,Y 448.045,Z 304.182,A -85,B 0,C 180,E1 20930.246,E2 20930.246} C_VEL
LIN {X 0,Y 440.31,Z 288.064,A -85,B 0,C 180,E1 20926.881,E2 20926.881} C_VEL
LIN {X 0,Y 435.143,Z 278.319,A -85,B 0,C 180,E1 20924.577,E2 20924.577} C_VEL
LIN {X 0,Y 432.867,Z 273.988,A -85,B 0,C 180,E1 20923.499,E2 20923.499} C_VEL
LIN {X 0,Y 430.488,Z 269.522,A -85,B 0,C 180,E1 20922.343,E2 20922.343} C_VEL
LIN {X 0,Y 428.418,Z 265.876,A -85,B 0,C 180,E1 20921.337,E2 20921.337} C_VEL
LIN {X 0,Y 427.717,Z 264.514,A -85,B 0,C 180,E1 20920.968,E2 20920.968} C_VEL
LIN {X 0,Y 425.754,Z 261.51,A -85,B 0,C 180,E1 20920.04,E2 20920.04} C_VEL
LIN {X 0,Y 425.307,Z 259.744,A -85,B 0,C 180,E1 20919.625,E2 20919.625} C_VEL
LIN {X 0,Y 425.31,Z 259.74,A -85,B 0,C 180,E1 20915.8,E2 20915.8} C_VEL
LIN {X 0,Y 425.347,Z 260.011,A -85,B 0,C 180,E1 20914.468,E2 20914.468} C_VEL
LIN {X 0,Y 434.01,Z 285.31,A -85,B 0,C 180,E1 20911.526,E2 20911.526} C_VEL
LIN {X 0,Y 436.813,Z 294.933,A -85,B 0,C 180,E1 20910.465,E2 20910.465} C_VEL
LIN {X 0,Y 435.625,Z 337.524,A -85,B 0,C 180,E1 20906.736,E2 20906.736} C_VEL
LIN {X 0,Y 434.352,Z 379.151,A -85,B 0,C 180,E1 20903.11,E2 20903.11} C_VEL
LIN {X 0,Y 432.896,Z 423.131,A -85,B 0,C 180,E1 20899.287,E2 20899.287} C_VEL
LIN {X 0,Y 432.011,Z 453.534,A -85,B 0,C 180,E1 20896.691,E2 20896.691} C_VEL
LIN {X 0,Y 429.822,Z 597.476,A -85,B 0,C 180,E1 20893.924,E2 20893.924} C_VEL
LIN {X 0,Y 429.624,Z 614.188,A -85,B 0,C 180,E1 20893.36,E2 20893.36} C_VEL
LIN {X 0,Y 429.227,Z 630.106,A -85,B 0,C 180,E1 20892.567,E2 20892.567} C_VEL
LIN {X 0,Y 428.729,Z 645.085,A -85,B 0,C 180,E1 20891.57,E2 20891.57} C_VEL
LIN {X 0,Y 428.117,Z 659.864,A -85,B 0,C 180,E1 20890.292,E2 20890.292} C_VEL
LIN {X 0,Y 427.503,Z 672.769,A -85,B 0,C 180,E1 20888.88,E2 20888.88} C_VEL
LIN {X 0,Y 426.907,Z 684.632,A -85,B 0,C 180,E1 20887.266,E2 20887.266} C_VEL
LIN {X 0,Y 426.382,Z 694.826,A -85,B 0,C 180,E1 20885.518,E2 20885.518} C_VEL
LIN {X 0,Y 425.985,Z 703.539,A -85,B 0,C 180,E1 20883.634,E2 20883.634} C_VEL
LIN {X 0,Y 425.701,Z 710.666,A -85,B 0,C 180,E1 20881.616,E2 20881.616} C_VEL
LIN {X 0,Y 425.538,Z 715.851,A -85,B 0,C 180,E1 20879.597,E2 20879.597} C_VEL
LIN {X 0,Y 425.475,Z 719.484,A -85,B 0,C 180,E1 20877.441,E2 20877.441} C_VEL
LIN {X 0,Y 425.509,Z 721.181,A -85,B 0,C 180,E1 20875.283,E2 20875.283} C_VEL
LIN {X 0,Y 425.62,Z 721.136,A -85,B 0,C 180,E1 20873.255,E2 20873.255} C_VEL
LIN {X 0,Y 425.795,Z 719.343,A -85,B 0,C 180,E1 20871.221,E2 20871.221} C_VEL
LIN {X 0,Y 426.09,Z 715.841,A -85,B 0,C 180,E1 20869.18,E2 20869.18} C_VEL
LIN {X 0,Y 426.457,Z 710.36,A -85,B 0,C 180,E1 20867.131,E2 20867.131} C_VEL
LIN {X 0,Y 426.945,Z 703.271,A -85,B 0,C 180,E1 20865.211,E2 20865.211} C_VEL
LIN {X 0,Y 427.502,Z 694.54,A -85,B 0,C 180,E1 20863.421,E2 20863.421} C_VEL
LIN {X 0,Y 428.088,Z 684.696,A -85,B 0,C 180,E1 20861.832,E2 20861.832} C_VEL
LIN {X 0,Y 428.723,Z 672.787,A -85,B 0,C 180,E1 20860.306,E2 20860.306} C_VEL
LIN {X 0,Y 429.25,Z 660.691,A -85,B 0,C 180,E1 20859.077,E2 20859.077} C_VEL
LIN {X 0,Y 429.724,Z 646.315,A -85,B 0,C 180,E1 20857.929,E2 20857.929} C_VEL
LIN {X 0,Y 430.042,Z 630.969,A -85,B 0,C 180,E1 20857.008,E2 20857.008} C_VEL
LIN {X 0,Y 430.206,Z 615.329,A -85,B 0,C 180,E1 20856.33,E2 20856.33} C_VEL
LIN {X 0,Y 430.157,Z 598.02,A -85,B 0,C 180,E1 20855.852,E2 20855.852} C_VEL
LIN {X 0,Y 431.366,Z 524.079,A -85,B 0,C 180,E1 20854.375,E2 20854.375} C_VEL
LIN {X 0,Y 432.973,Z 466.962,A -85,B 0,C 180,E1 20853.126,E2 20853.126} C_VEL
LIN {X 0,Y 434.848,Z 456.606,A -85,B 0,C 180,E1 20852.399,E2 20852.399} C_VEL
LIN {X 0,Y 435.785,Z 415.807,A -85,B 0,C 180,E1 20849.074,E2 20849.074} C_VEL
LIN {X 0,Y 436.373,Z 379.096,A -85,B 0,C 180,E1 20846.167,E2 20846.167} C_VEL
LIN {X 0,Y 436.505,Z 376.01,A -85,B 0,C 180,E1 20845.901,E2 20845.901} C_VEL
LIN {X 0,Y 438.909,Z 376.309,A -85,B 0,C 180,E1 20845.554,E2 20845.554} C_VEL
LIN {X 0,Y 442.441,Z 374.706,A -85,B 0,C 180,E1 20845.247,E2 20845.247} C_VEL
LIN {X 0,Y 447.088,Z 373.556,A -85,B 0,C 180,E1 20844.762,E2 20844.762} C_VEL
LIN {X 0,Y 449.628,Z 372.711,A -85,B 0,C 180,E1 20844.522,E2 20844.522} C_VEL
LIN {X 0,Y 457.524,Z 370.458,A -85,B 0,C 180,E1 20843.767,E2 20843.767} C_VEL
LIN {X 0,Y 458.879,Z 388.867,A -85,B 0,C 180,E1 20842.009,E2 20842.009} C_VEL
LIN {X 0,Y 462.148,Z 405.463,A -85,B 0,C 180,E1 20840.26,E2 20840.26} C_VEL
LIN {X 0,Y 467.098,Z 419.868,A -85,B 0,C 180,E1 20838.591,E2 20838.591} C_VEL
LIN {X 0,Y 474.337,Z 433.686,A -85,B 0,C 180,E1 20836.831,E2 20836.831} C_VEL
LIN {X 0,Y 482.805,Z 445.012,A -85,B 0,C 180,E1 20835.242,E2 20835.242} C_VEL
LIN {X 0,Y 492.638,Z 454.774,A -85,B 0,C 180,E1 20833.736,E2 20833.736} C_VEL
LIN {X 0,Y 498.882,Z 459.831,A -85,B 0,C 180,E1 20832.897,E2 20832.897} C_VEL
LIN {X 0,Y 485.805,Z 480.948,A -85,B 0,C 180,E1 20832.388,E2 20832.388} C_VEL
LIN {X 0,Y 476.697,Z 498.137,A -85,B 0,C 180,E1 20831.836,E2 20831.836} C_VEL
LIN {X 0,Y 470.688,Z 511.002,A -85,B 0,C 180,E1 20831.349,E2 20831.349} C_VEL
LIN {X 0,Y 462.657,Z 527.357,A -85,B 0,C 180,E1 20830.743,E2 20830.743} C_VEL
LIN {X 0,Y 454.93,Z 547.329,A -85,B 0,C 180,E1 20829.862,E2 20829.862} C_VEL
LIN {X 0,Y 452.701,Z 569.04,A -85,B 0,C 180,E1 20829.646,E2 20829.646} C_VEL
LIN {X 0,Y 451.623,Z 597.738,A -85,B 0,C 180,E1 20829.096,E2 20829.096} C_VEL
LIN {X 0,Y 449.722,Z 623.27,A -85,B 0,C 180,E1 20828.392,E2 20828.392} C_VEL
LIN {X 0,Y 447.648,Z 647.121,A -85,B 0,C 180,E1 20827.492,E2 20827.492} C_VEL
LIN {X 0,Y 445.398,Z 669.706,A -85,B 0,C 180,E1 20826.399,E2 20826.399} C_VEL
LIN {X 0,Y 442.97,Z 691.584,A -85,B 0,C 180,E1 20825.077,E2 20825.077} C_VEL
LIN {X 0,Y 440.416,Z 712.534,A -85,B 0,C 180,E1 20823.539,E2 20823.539} C_VEL
LIN {X 0,Y 437.887,Z 731.897,A -85,B 0,C 180,E1 20821.834,E2 20821.834} C_VEL
LIN {X 0,Y 435.51,Z 749.168,A -85,B 0,C 180,E1 20820.033,E2 20820.033} C_VEL
LIN {X 0,Y 432.915,Z 766.973,A -85,B 0,C 180,E1 20817.81,E2 20817.81} C_VEL
LIN {X 0,Y 430.711,Z 782.062,A -85,B 0,C 180,E1 20815.581,E2 20815.581} C_VEL
LIN {X 0,Y 428.704,Z 796.573,A -85,B 0,C 180,E1 20813.068,E2 20813.068} C_VEL
LIN {X 0,Y 426.989,Z 810.118,A -85,B 0,C 180,E1 20810.277,E2 20810.277} C_VEL
LIN {X 0,Y 425.689,Z 821.861,A -85,B 0,C 180,E1 20807.355,E2 20807.355} C_VEL
LIN {X 0,Y 424.86,Z 831.042,A -85,B 0,C 180,E1 20804.585,E2 20804.585} C_VEL
LIN {X 0,Y 424.356,Z 838.482,A -85,B 0,C 180,E1 20801.829,E2 20801.829} C_VEL
LIN {X 0,Y 424.049,Z 844.73,A -85,B 0,C 180,E1 20798.816,E2 20798.816} C_VEL
LIN {X 0,Y 423.942,Z 848.937,A -85,B 0,C 180,E1 20795.956,E2 20795.956} C_VEL
LIN {X 0,Y 423.914,Z 851.522,A -85,B 0,C 180,E1 20793.11,E2 20793.11} C_VEL
LIN {X 0,Y 423.908,Z 852.465,A -85,B 0,C 180,E1 20790.135,E2 20790.135} C_VEL
LIN {X 0,Y 423.91,Z 851.739,A -85,B 0,C 180,E1 20787.296,E2 20787.296} C_VEL
LIN {X 0,Y 423.937,Z 849.421,A -85,B 0,C 180,E1 20784.451,E2 20784.451} C_VEL
LIN {X 0,Y 424.043,Z 845.202,A -85,B 0,C 180,E1 20781.457,E2 20781.457} C_VEL
LIN {X 0,Y 424.298,Z 839.422,A -85,B 0,C 180,E1 20778.583,E2 20778.583} C_VEL
LIN {X 0,Y 424.798,Z 831.857,A -85,B 0,C 180,E1 20775.691,E2 20775.691} C_VEL
LIN {X 0,Y 425.638,Z 822.34,A -85,B 0,C 180,E1 20772.783,E2 20772.783} C_VEL
LIN {X 0,Y 426.915,Z 810.664,A -85,B 0,C 180,E1 20769.862,E2 20769.862} C_VEL
LIN {X 0,Y 428.533,Z 797.698,A -85,B 0,C 180,E1 20767.163,E2 20767.163} C_VEL
LIN {X 0,Y 430.458,Z 783.693,A -85,B 0,C 180,E1 20764.698,E2 20764.698} C_VEL
LIN {X 0,Y 432.754,Z 767.869,A -85,B 0,C 180,E1 20762.328,E2 20762.328} C_VEL
LIN {X 0,Y 435.13,Z 751.339,A -85,B 0,C 180,E1 20760.242,E2 20760.242} C_VEL
LIN {X 0,Y 437.483,Z 734.506,A -85,B 0,C 180,E1 20758.441,E2 20758.441} C_VEL
LIN {X 0,Y 439.885,Z 715.934,A -85,B 0,C 180,E1 20756.768,E2 20756.768} C_VEL
LIN {X 0,Y 442.441,Z 695.419,A -85,B 0,C 180,E1 20755.206,E2 20755.206} C_VEL
LIN {X 0,Y 444.889,Z 673.883,A -85,B 0,C 180,E1 20753.846,E2 20753.846} C_VEL
LIN {X 0,Y 447.35,Z 650.149,A -85,B 0,C 180,E1 20752.645,E2 20752.645} C_VEL
LIN {X 0,Y 449.591,Z 625.483,A -85,B 0,C 180,E1 20751.671,E2 20751.671} C_VEL
LIN {X 0,Y 451.516,Z 600.691,A -85,B 0,C 180,E1 20750.96,E2 20750.96} C_VEL
LIN {X 0,Y 452.665,Z 574.453,A -85,B 0,C 180,E1 20750.415,E2 20750.415} C_VEL
LIN {X 0,Y 453.772,Z 560.316,A -85,B 0,C 180,E1 20750.243,E2 20750.243} C_VEL
LIN {X 0,Y 455.65,Z 546.841,A -85,B 0,C 180,E1 20750.152,E2 20750.152} C_VEL
LIN {X 0,Y 465.255,Z 527.222,A -85,B 0,C 180,E1 20749.153,E2 20749.153} C_VEL
LIN {X 0,Y 474.325,Z 512.416,A -85,B 0,C 180,E1 20748.555,E2 20748.555} C_VEL
LIN {X 0,Y 478.943,Z 504.712,A -85,B 0,C 180,E1 20748.244,E2 20748.244} C_VEL
LIN {X 0,Y 488.907,Z 489.094,A -85,B 0,C 180,E1 20747.673,E2 20747.673} C_VEL
LIN {X 0,Y 488.866,Z 488.654,A -85,B 0,C 180,E1 20747.634,E2 20747.634} C_VEL
LIN {X 0,Y 478.77,Z 479.518,A -85,B 0,C 180,E1 20746.095,E2 20746.095} C_VEL
LIN {X 0,Y 470.025,Z 468.693,A -85,B 0,C 180,E1 20744.416,E2 20744.416} C_VEL
LIN {X 0,Y 463.535,Z 457.434,A -85,B 0,C 180,E1 20742.801,E2 20742.801} C_VEL
LIN {X 0,Y 458.359,Z 444.185,A -85,B 0,C 180,E1 20741.04,E2 20741.04} C_VEL
LIN {X 0,Y 454.972,Z 428.942,A -85,B 0,C 180,E1 20739.184,E2 20739.184} C_VEL
LIN {X 0,Y 453.541,Z 412.226,A -85,B 0,C 180,E1 20737.319,E2 20737.319} C_VEL
LIN {X 0,Y 454.131,Z 393.8,A -85,B 0,C 180,E1 20735.449,E2 20735.449} C_VEL
LIN {X 0,Y 460.646,Z 343.523,A -85,B 0,C 180,E1 20730.734,E2 20730.734} C_VEL
LIN {X 0,Y 461.826,Z 335.207,A -85,B 0,C 180,E1 20729.936,E2 20729.936} C_VEL
LIN {X 0,Y 449.914,Z 339.72,A -85,B 0,C 180,E1 20728.618,E2 20728.618} C_VEL
LIN {X 0,Y 445.442,Z 341.429,A -85,B 0,C 180,E1 20728.097,E2 20728.097} C_VEL
LIN {X 0,Y 441.623,Z 343.005,A -85,B 0,C 180,E1 20727.654,E2 20727.654} C_VEL
LIN {X 0,Y 440.166,Z 343.439,A -85,B 0,C 180,E1 20727.459,E2 20727.459} C_VEL
LIN {X 0,Y 436.828,Z 345.108,A -85,B 0,C 180,E1 20727.096,E2 20727.096} C_VEL
LIN {X 0,Y 434.902,Z 345.07,A -85,B 0,C 180,E1 20726.746,E2 20726.746} C_VEL
LIN {X 0,Y 434.487,Z 387.423,A -85,B 0,C 180,E1 20723.666,E2 20723.666} C_VEL
LIN {X 0,Y 433.793,Z 429.731,A -85,B 0,C 180,E1 20720.508,E2 20720.508} C_VEL
LIN {X 0,Y 432.806,Z 473.993,A -85,B 0,C 180,E1 20717.13,E2 20717.13} C_VEL
LIN {X 0,Y 431.991,Z 503.719,A -85,B 0,C 180,E1 20714.822,E2 20714.822} C_VEL
LIN {X 0,Y 430.558,Z 512.852,A -85,B 0,C 180,E1 20714.224,E2 20714.224} C_VEL
LIN {X 0,Y 428.877,Z 612.258,A -85,B 0,C 180,E1 20712.252,E2 20712.252} C_VEL
LIN {X 0,Y 428.972,Z 629.494,A -85,B 0,C 180,E1 20711.836,E2 20711.836} C_VEL
LIN {X 0,Y 428.92,Z 643.571,A -85,B 0,C 180,E1 20711.258,E2 20711.258} C_VEL
LIN {X 0,Y 428.697,Z 656.847,A -85,B 0,C 180,E1 20710.481,E2 20710.481} C_VEL
LIN {X 0,Y 428.324,Z 670.391,A -85,B 0,C 180,E1 20709.404,E2 20709.404} C_VEL
LIN {X 0,Y 427.861,Z 682.562,A -85,B 0,C 180,E1 20708.127,E2 20708.127} C_VEL
LIN {X 0,Y 427.366,Z 692.936,A -85,B 0,C 180,E1 20706.717,E2 20706.717} C_VEL
LIN {X 0,Y 426.904,Z 701.444,A -85,B 0,C 180,E1 20705.24,E2 20705.24} C_VEL
LIN {X 0,Y 426.474,Z 708.64,A -85,B 0,C 180,E1 20703.629,E2 20703.629} C_VEL
LIN {X 0,Y 426.082,Z 714.772,A -85,B 0,C 180,E1 20701.748,E2 20701.748} C_VEL
LIN {X 0,Y 425.795,Z 718.876,A -85,B 0,C 180,E1 20699.865,E2 20699.865} C_VEL
LIN {X 0,Y 425.618,Z 721.177,A -85,B 0,C 180,E1 20697.98,E2 20697.98} C_VEL
LIN {X 0,Y 425.499,Z 721.733,A -85,B 0,C 180,E1 20695.957,E2 20695.957} C_VEL
LIN {X 0,Y 425.474,Z 720.318,A -85,B 0,C 180,E1 20693.929,E2 20693.929} C_VEL
LIN {X 0,Y 425.532,Z 716.916,A -85,B 0,C 180,E1 20691.895,E2 20691.895} C_VEL
LIN {X 0,Y 425.7,Z 711.801,A -85,B 0,C 180,E1 20689.99,E2 20689.99} C_VEL
LIN {X 0,Y 425.96,Z 705.029,A -85,B 0,C 180,E1 20688.191,E2 20688.191} C_VEL
LIN {X 0,Y 426.313,Z 697.048,A -85,B 0,C 180,E1 20686.573,E2 20686.573} C_VEL
LIN {X 0,Y 426.764,Z 686.542,A -85,B 0,C 180,E1 20684.926,E2 20684.926} C_VEL
LIN {X 0,Y 427.247,Z 674.634,A -85,B 0,C 180,E1 20683.48,E2 20683.48} C_VEL
LIN {X 0,Y 427.693,Z 661.564,A -85,B 0,C 180,E1 20682.255,E2 20682.255} C_VEL
LIN {X 0,Y 428.078,Z 647.986,A -85,B 0,C 180,E1 20681.288,E2 20681.288} C_VEL
LIN {X 0,Y 428.326,Z 633.619,A -85,B 0,C 180,E1 20680.54,E2 20680.54} C_VEL
LIN {X 0,Y 428.437,Z 618.515,A -85,B 0,C 180,E1 20680.016,E2 20680.016} C_VEL
LIN {X 0,Y 429.966,Z 502.584,A -85,B 0,C 180,E1 20677.797,E2 20677.797} C_VEL
LIN {X 0,Y 430.918,Z 477.994,A -85,B 0,C 180,E1 20675.824,E2 20675.824} C_VEL
LIN {X 0,Y 432.379,Z 429.525,A -85,B 0,C 180,E1 20671.907,E2 20671.907} C_VEL
LIN {X 0,Y 433.802,Z 383.738,A -85,B 0,C 180,E1 20668.204,E2 20668.204} C_VEL
LIN {X 0,Y 435.11,Z 339.63,A -85,B 0,C 180,E1 20664.613,E2 20664.613} C_VEL
LIN {X 0,Y 436.356,Z 297.32,A -85,B 0,C 180,E1 20661.155,E2 20661.155} C_VEL
LIN {X 0,Y 438.053,Z 297.174,A -85,B 0,C 180,E1 20660.783,E2 20660.783} C_VEL
LIN {X 0,Y 440.628,Z 296.085,A -85,B 0,C 180,E1 20660.384,E2 20660.384} C_VEL
LIN {X 0,Y 444.025,Z 295.927,A -85,B 0,C 180,E1 20659.654,E2 20659.654} C_VEL
LIN {X 0,Y 448.677,Z 306.057,A -85,B 0,C 180,E1 20657.006,E2 20657.006} C_VEL
LIN {X 0,Y 453.684,Z 317.863,A -85,B 0,C 180,E1 20654.253,E2 20654.253} C_VEL
LIN {X 0,Y 456.531,Z 325.433,A -85,B 0,C 180,E1 20652.667,E2 20652.667} C_VEL
LIN {X 0,Y 455.215,Z 335.071,A -85,B 0,C 180,E1 20651.591,E2 20651.591} C_VEL
LIN {X 0,Y 455.686,Z 338.147,A -85,B 0,C 180,E1 20651.473,E2 20651.473} C_VEL
LIN {X 0,Y 453.123,Z 417.93,A -85,B 0,C 180,E1 20650.036,E2 20650.036} C_VEL
LIN {X 0,Y 452.998,Z 420.902,A -85,B 0,C 180,E1 20649.979,E2 20649.979} C_VEL
LIN {X 0,Y 451.906,Z 428.577,A -85,B 0,C 180,E1 20649.915,E2 20649.915} C_VEL
LIN {X 0,Y 446.241,Z 449.037,A -85,B 0,C 180,E1 20650.027,E2 20650.027} C_VEL
LIN {X 0,Y 445.359,Z 455.61,A -85,B 0,C 180,E1 20649.952,E2 20649.952} C_VEL
LIN {X 0,Y 440.679,Z 541.324,A -85,B 0,C 180,E1 20648.031,E2 20648.031} C_VEL
LIN {X 0,Y 438.386,Z 582.629,A -85,B 0,C 180,E1 20646.977,E2 20646.977} C_VEL
LIN {X 0,Y 436.902,Z 603.51,A -85,B 0,C 180,E1 20646.189,E2 20646.189} C_VEL
LIN {X 0,Y 435.023,Z 624.252,A -85,B 0,C 180,E1 20645.129,E2 20645.129} C_VEL
LIN {X 0,Y 432.935,Z 643.169,A -85,B 0,C 180,E1 20643.9,E2 20643.9} C_VEL
LIN {X 0,Y 430.635,Z 661.462,A -85,B 0,C 180,E1 20642.435,E2 20642.435} C_VEL
LIN {X 0,Y 428.154,Z 679.506,A -85,B 0,C 180,E1 20640.681,E2 20640.681} C_VEL
LIN {X 0,Y 425.703,Z 696.336,A -85,B 0,C 180,E1 20638.706,E2 20638.706} C_VEL
LIN {X 0,Y 423.523,Z 711.016,A -85,B 0,C 180,E1 20636.651,E2 20636.651} C_VEL
LIN {X 0,Y 421.506,Z 724.73,A -85,B 0,C 180,E1 20634.37,E2 20634.37} C_VEL
LIN {X 0,Y 419.806,Z 736.874,A -85,B 0,C 180,E1 20631.958,E2 20631.958} C_VEL
LIN {X 0,Y 418.445,Z 747.584,A -85,B 0,C 180,E1 20629.399,E2 20629.399} C_VEL
LIN {X 0,Y 417.474,Z 756.334,A -85,B 0,C 180,E1 20626.846,E2 20626.846} C_VEL
LIN {X 0,Y 416.803,Z 763.715,A -85,B 0,C 180,E1 20624.163,E2 20624.163} C_VEL
LIN {X 0,Y 416.401,Z 769.619,A -85,B 0,C 180,E1 20621.356,E2 20621.356} C_VEL
LIN {X 0,Y 416.209,Z 773.752,A -85,B 0,C 180,E1 20618.566,E2 20618.566} C_VEL
LIN {X 0,Y 416.132,Z 776.184,A -85,B 0,C 180,E1 20615.875,E2 20615.875} C_VEL
LIN {X 0,Y 416.108,Z 777.074,A -85,B 0,C 180,E1 20613.03,E2 20613.03} C_VEL
LIN {X 0,Y 416.12,Z 776.282,A -85,B 0,C 180,E1 20610.275,E2 20610.275} C_VEL
LIN {X 0,Y 416.191,Z 773.918,A -85,B 0,C 180,E1 20607.522,E2 20607.522} C_VEL
LIN {X 0,Y 416.379,Z 769.941,A -85,B 0,C 180,E1 20604.764,E2 20604.764} C_VEL
LIN {X 0,Y 416.747,Z 764.26,A -85,B 0,C 180,E1 20602.001,E2 20602.001} C_VEL
LIN {X 0,Y 417.372,Z 757.175,A -85,B 0,C 180,E1 20599.37,E2 20599.37} C_VEL
LIN {X 0,Y 418.32,Z 748.268,A -85,B 0,C 180,E1 20596.735,E2 20596.735} C_VEL
LIN {X 0,Y 419.678,Z 737.283,A -85,B 0,C 180,E1 20594.099,E2 20594.099} C_VEL
LIN {X 0,Y 421.379,Z 724.673,A -85,B 0,C 180,E1 20591.604,E2 20591.604} C_VEL
LIN {X 0,Y 423.285,Z 711.317,A -85,B 0,C 180,E1 20589.393,E2 20589.393} C_VEL
LIN {X 0,Y 425.488,Z 695.982,A -85,B 0,C 180,E1 20587.259,E2 20587.259} C_VEL
LIN {X 0,Y 427.8,Z 679.522,A -85,B 0,C 180,E1 20585.342,E2 20585.342} C_VEL
LIN {X 0,Y 430.137,Z 661.979,A -85,B 0,C 180,E1 20583.642,E2 20583.642} C_VEL
LIN {X 0,Y 432.394,Z 643.368,A -85,B 0,C 180,E1 20582.154,E2 20582.154} C_VEL
LIN {X 0,Y 434.508,Z 623.592,A -85,B 0,C 180,E1 20580.877,E2 20580.877} C_VEL
LIN {X 0,Y 436.289,Z 603.029,A -85,B 0,C 180,E1 20579.837,E2 20579.837} C_VEL
LIN {X 0,Y 437.717,Z 582.055,A -85,B 0,C 180,E1 20579.053,E2 20579.053} C_VEL
LIN {X 0,Y 440.124,Z 536.724,A -85,B 0,C 180,E1 20577.918,E2 20577.918} C_VEL
LIN {X 0,Y 444.546,Z 451.293,A -85,B 0,C 180,E1 20576.033,E2 20576.033} C_VEL
LIN {X 0,Y 447.413,Z 378.746,A -85,B 0,C 180,E1 20574.636,E2 20574.636} C_VEL
LIN {X 0,Y 448.818,Z 334.09,A -85,B 0,C 180,E1 20573.837,E2 20573.837} C_VEL
LIN {X 0,Y 449.741,Z 326.405,A -85,B 0,C 180,E1 20573.111,E2 20573.111} C_VEL
LIN {X 0,Y 442.486,Z 309.613,A -85,B 0,C 180,E1 20569.998,E2 20569.998} C_VEL
LIN {X 0,Y 435.203,Z 294.19,A -85,B 0,C 180,E1 20566.744,E2 20566.744} C_VEL
LIN {X 0,Y 430.108,Z 284.4,A -85,B 0,C 180,E1 20564.406,E2 20564.406} C_VEL
LIN {X 0,Y 427.347,Z 279.303,A -85,B 0,C 180,E1 20563.094,E2 20563.094} C_VEL
LIN {X 0,Y 425.133,Z 275.169,A -85,B 0,C 180,E1 20561.996,E2 20561.996} C_VEL
LIN {X 0,Y 422.747,Z 270.661,A -85,B 0,C 180,E1 20560.752,E2 20560.752} C_VEL
LIN {X 0,Y 420.738,Z 267.329,A -85,B 0,C 180,E1 20559.738,E2 20559.738} C_VEL
LIN {X 0,Y 419.989,Z 265.735,A -85,B 0,C 180,E1 20559.292,E2 20559.292} C_VEL
LIN {X 0,Y 417.95,Z 262.847,A -85,B 0,C 180,E1 20558.288,E2 20558.288} C_VEL
LIN {X 0,Y 417.381,Z 260.726,A -85,B 0,C 180,E1 20557.764,E2 20557.764} C_VEL
LIN {X 0,Y 417.38,Z 260.772,A -85,B 0,C 180,E1 20555.032,E2 20555.032} C_VEL
LIN {X 0,Y 426.418,Z 287.122,A -85,B 0,C 180,E1 20551.917,E2 20551.917} C_VEL
LIN {X 0,Y 429.468,Z 297.671,A -85,B 0,C 180,E1 20550.741,E2 20550.741} C_VEL
LIN {X 0,Y 428.245,Z 339.157,A -85,B 0,C 180,E1 20547.084,E2 20547.084} C_VEL
LIN {X 0,Y 426.843,Z 381.986,A -85,B 0,C 180,E1 20543.321,E2 20543.321} C_VEL
LIN {X 0,Y 425.351,Z 425.747,A -85,B 0,C 180,E1 20539.5,E2 20539.5} C_VEL
LIN {X 0,Y 424.461,Z 454.581,A -85,B 0,C 180,E1 20537.019,E2 20537.019} C_VEL
LIN {X 0,Y 422.08,Z 598.502,A -85,B 0,C 180,E1 20534.175,E2 20534.175} C_VEL
LIN {X 0,Y 421.877,Z 615.061,A -85,B 0,C 180,E1 20533.609,E2 20533.609} C_VEL
LIN {X 0,Y 421.465,Z 631.176,A -85,B 0,C 180,E1 20532.795,E2 20532.795} C_VEL
LIN {X 0,Y 420.952,Z 646.13,A -85,B 0,C 180,E1 20531.787,E2 20531.787} C_VEL
LIN {X 0,Y 420.306,Z 661.299,A -85,B 0,C 180,E1 20530.455,E2 20530.455} C_VEL
LIN {X 0,Y 419.68,Z 673.945,A -85,B 0,C 180,E1 20529.047,E2 20529.047} C_VEL
LIN {X 0,Y 419.061,Z 685.876,A -85,B 0,C 180,E1 20527.403,E2 20527.403} C_VEL
LIN {X 0,Y 418.518,Z 696.119,A -85,B 0,C 180,E1 20525.622,E2 20525.622} C_VEL
LIN {X 0,Y 418.133,Z 704.344,A -85,B 0,C 180,E1 20523.84,E2 20523.84} C_VEL
LIN {X 0,Y 417.827,Z 711.622,A -85,B 0,C 180,E1 20521.783,E2 20521.783} C_VEL
LIN {X 0,Y 417.656,Z 716.975,A -85,B 0,C 180,E1 20519.726,E2 20519.726} C_VEL
LIN {X 0,Y 417.587,Z 720.724,A -85,B 0,C 180,E1 20517.53,E2 20517.53} C_VEL
LIN {X 0,Y 417.621,Z 722.497,A -85,B 0,C 180,E1 20515.469,E2 20515.469} C_VEL
LIN {X 0,Y 417.751,Z 722.591,A -85,B 0,C 180,E1 20513.265,E2 20513.265} C_VEL
LIN {X 0,Y 417.947,Z 720.896,A -85,B 0,C 180,E1 20511.193,E2 20511.193} C_VEL
LIN {X 0,Y 418.27,Z 717.464,A -85,B 0,C 180,E1 20509.115,E2 20509.115} C_VEL
LIN {X 0,Y 418.644,Z 712.478,A -85,B 0,C 180,E1 20507.167,E2 20507.167} C_VEL
LIN {X 0,Y 419.152,Z 705.569,A -85,B 0,C 180,E1 20505.213,E2 20505.213} C_VEL
LIN {X 0,Y 419.75,Z 697.075,A -85,B 0,C 180,E1 20503.391,E2 20503.391} C_VEL
LIN {X 0,Y 420.407,Z 687.042,A -85,B 0,C 180,E1 20501.704,E2 20501.704} C_VEL
LIN {X 0,Y 421.065,Z 675.24,A -85,B 0,C 180,E1 20500.15,E2 20500.15} C_VEL
LIN {X 0,Y 421.673,Z 662.302,A -85,B 0,C 180,E1 20498.802,E2 20498.802} C_VEL
LIN {X 0,Y 422.168,Z 648.315,A -85,B 0,C 180,E1 20497.659,E2 20497.659} C_VEL
LIN {X 0,Y 422.514,Z 633.121,A -85,B 0,C 180,E1 20496.722,E2 20496.722} C_VEL
LIN {X 0,Y 422.687,Z 617.23,A -85,B 0,C 180,E1 20496.016,E2 20496.016} C_VEL
LIN {X 0,Y 422.64,Z 599.621,A -85,B 0,C 180,E1 20495.516,E2 20495.516} C_VEL
LIN {X 0,Y 423.936,Z 528.275,A -85,B 0,C 180,E1 20494.032,E2 20494.032} C_VEL
LIN {X 0,Y 425.816,Z 468.892,A -85,B 0,C 180,E1 20492.674,E2 20492.674} C_VEL
LIN {X 0,Y 427.84,Z 457.907,A -85,B 0,C 180,E1 20491.907,E2 20491.907} C_VEL
LIN {X 0,Y 428.896,Z 416.703,A -85,B 0,C 180,E1 20488.521,E2 20488.521} C_VEL
LIN {X 0,Y 429.602,Z 384.969,A -85,B 0,C 180,E1 20485.963,E2 20485.963} C_VEL
LIN {X 0,Y 431.999,Z 385.206,A -85,B 0,C 180,E1 20485.617,E2 20485.617} C_VEL
LIN {X 0,Y 435.284,Z 383.761,A -85,B 0,C 180,E1 20485.32,E2 20485.32} C_VEL
LIN {X 0,Y 440.628,Z 382.208,A -85,B 0,C 180,E1 20484.776,E2 20484.776} C_VEL
LIN {X 0,Y 443.177,Z 381.343,A -85,B 0,C 180,E1 20484.534,E2 20484.534} C_VEL
LIN {X 0,Y 451.375,Z 378.895,A -85,B 0,C 180,E1 20483.75,E2 20483.75} C_VEL
LIN {X 0,Y 453.189,Z 397.18,A -85,B 0,C 180,E1 20481.928,E2 20481.928} C_VEL
LIN {X 0,Y 456.932,Z 413.635,A -85,B 0,C 180,E1 20480.123,E2 20480.123} C_VEL
LIN {X 0,Y 462.386,Z 427.869,A -85,B 0,C 180,E1 20478.406,E2 20478.406} C_VEL
LIN {X 0,Y 469.574,Z 440.742,A -85,B 0,C 180,E1 20476.715,E2 20476.715} C_VEL
LIN {X 0,Y 478.505,Z 452.183,A -85,B 0,C 180,E1 20475.068,E2 20475.068} C_VEL
LIN {X 0,Y 488.468,Z 461.714,A -85,B 0,C 180,E1 20473.564,E2 20473.564} C_VEL
LIN {X 0,Y 489.76,Z 462.831,A -85,B 0,C 180,E1 20473.383,E2 20473.383} C_VEL
LIN {X 0,Y 477.646,Z 482.923,A -85,B 0,C 180,E1 20472.869,E2 20472.869} C_VEL
LIN {X 0,Y 468.837,Z 500.116,A -85,B 0,C 180,E1 20472.288,E2 20472.288} C_VEL
LIN {X 0,Y 464.523,Z 509.293,A -85,B 0,C 180,E1 20471.939,E2 20471.939} C_VEL
LIN {X 0,Y 456.438,Z 525.622,A -85,B 0,C 180,E1 20471.335,E2 20471.335} C_VEL
LIN {X 0,Y 448.835,Z 544.984,A -85,B 0,C 180,E1 20470.481,E2 20470.481} C_VEL
LIN {X 0,Y 446.496,Z 565.578,A -85,B 0,C 180,E1 20470.295,E2 20470.295} C_VEL
LIN {X 0,Y 445.306,Z 593.199,A -85,B 0,C 180,E1 20469.786,E2 20469.786} C_VEL
LIN {X 0,Y 443.463,Z 618.519,A -85,B 0,C 180,E1 20469.11,E2 20469.11} C_VEL
LIN {X 0,Y 441.206,Z 642.914,A -85,B 0,C 180,E1 20468.219,E2 20468.219} C_VEL
LIN {X 0,Y 438.858,Z 666.121,A -85,B 0,C 180,E1 20467.117,E2 20467.117} C_VEL
LIN {X 0,Y 436.343,Z 687.969,A -85,B 0,C 180,E1 20465.828,E2 20465.828} C_VEL
LIN {X 0,Y 433.704,Z 709.065,A -85,B 0,C 180,E1 20464.31,E2 20464.31} C_VEL
LIN {X 0,Y 430.996,Z 729.305,A -85,B 0,C 180,E1 20462.562,E2 20462.562} C_VEL
LIN {X 0,Y 428.48,Z 747.113,A -85,B 0,C 180,E1 20460.733,E2 20460.733} C_VEL
LIN {X 0,Y 425.933,Z 763.698,A -85,B 0,C 180,E1 20458.689,E2 20458.689} C_VEL
LIN {X 0,Y 423.618,Z 778.822,A -85,B 0,C 180,E1 20456.494,E2 20456.494} C_VEL
LIN {X 0,Y 421.273,Z 794.467,A -85,B 0,C 180,E1 20453.796,E2 20453.796} C_VEL
LIN {X 0,Y 419.364,Z 808.207,A -85,B 0,C 180,E1 20450.955,E2 20450.955} C_VEL
LIN {X 0,Y 418.039,Z 819.13,A -85,B 0,C 180,E1 20448.26,E2 20448.26} C_VEL
LIN {X 0,Y 417.077,Z 828.713,A -85,B 0,C 180,E1 20445.432,E2 20445.432} C_VEL
LIN {X 0,Y 416.413,Z 837.362,A -85,B 0,C 180,E1 20442.245,E2 20442.245} C_VEL
LIN {X 0,Y 416.098,Z 843.538,A -85,B 0,C 180,E1 20439.265,E2 20439.265} C_VEL
LIN {X 0,Y 415.97,Z 847.748,A -85,B 0,C 180,E1 20436.487,E2 20436.487} C_VEL
LIN {X 0,Y 415.937,Z 850.544,A -85,B 0,C 180,E1 20433.583,E2 20433.583} C_VEL
LIN {X 0,Y 415.934,Z 851.703,A -85,B 0,C 180,E1 20430.826,E2 20430.826} C_VEL
LIN {X 0,Y 415.937,Z 851.366,A -85,B 0,C 180,E1 20427.934,E2 20427.934} C_VEL
LIN {X 0,Y 415.952,Z 849.402,A -85,B 0,C 180,E1 20425.036,E2 20425.036} C_VEL
LIN {X 0,Y 416.021,Z 845.835,A -85,B 0,C 180,E1 20422.126,E2 20422.126} C_VEL
LIN {X 0,Y 416.247,Z 840.261,A -85,B 0,C 180,E1 20419.061,E2 20419.061} C_VEL
LIN {X 0,Y 416.7,Z 833.123,A -85,B 0,C 180,E1 20416.116,E2 20416.116} C_VEL
LIN {X 0,Y 417.464,Z 824.595,A -85,B 0,C 180,E1 20413.297,E2 20413.297} C_VEL
LIN {X 0,Y 418.687,Z 813.572,A -85,B 0,C 180,E1 20410.323,E2 20410.323} C_VEL
LIN {X 0,Y 420.33,Z 800.852,A -85,B 0,C 180,E1 20407.481,E2 20407.481} C_VEL
LIN {X 0,Y 422.298,Z 787.272,A -85,B 0,C 180,E1 20404.924,E2 20404.924} C_VEL
LIN {X 0,Y 424.678,Z 771.657,A -85,B 0,C 180,E1 20402.442,E2 20402.442} C_VEL
LIN {X 0,Y 427.269,Z 754.677,A -85,B 0,C 180,E1 20400.18,E2 20400.18} C_VEL
LIN {X 0,Y 429.778,Z 737.662,A -85,B 0,C 180,E1 20398.279,E2 20398.279} C_VEL
LIN {X 0,Y 432.558,Z 717.336,A -85,B 0,C 180,E1 20396.385,E2 20396.385} C_VEL
LIN {X 0,Y 435.1,Z 697.939,A -85,B 0,C 180,E1 20394.863,E2 20394.863} C_VEL
LIN {X 0,Y 437.789,Z 675.667,A -85,B 0,C 180,E1 20393.409,E2 20393.409} C_VEL
LIN {X 0,Y 440.366,Z 652.612,A -85,B 0,C 180,E1 20392.19,E2 20392.19} C_VEL
LIN {X 0,Y 442.687,Z 628.804,A -85,B 0,C 180,E1 20391.205,E2 20391.205} C_VEL
LIN {X 0,Y 444.926,Z 602.603,A -85,B 0,C 180,E1 20390.401,E2 20390.401} C_VEL
LIN {X 0,Y 446.239,Z 576.862,A -85,B 0,C 180,E1 20389.836,E2 20389.836} C_VEL
LIN {X 0,Y 447.242,Z 562.132,A -85,B 0,C 180,E1 20389.629,E2 20389.629} C_VEL
LIN {X 0,Y 449.713,Z 544.49,A -85,B 0,C 180,E1 20389.517,E2 20389.517} C_VEL
LIN {X 0,Y 459.169,Z 525.422,A -85,B 0,C 180,E1 20388.549,E2 20388.549} C_VEL
LIN {X 0,Y 468.74,Z 509.915,A -85,B 0,C 180,E1 20387.928,E2 20387.928} C_VEL
LIN {X 0,Y 479.942,Z 491.672,A -85,B 0,C 180,E1 20387.222,E2 20387.222} C_VEL
LIN {X 0,Y 470.108,Z 481.855,A -85,B 0,C 180,E1 20385.593,E2 20385.593} C_VEL
LIN {X 0,Y 461.306,Z 469.818,A -85,B 0,C 180,E1 20383.742,E2 20383.742} C_VEL
LIN {X 0,Y 454.523,Z 456.057,A -85,B 0,C 180,E1 20381.8,E2 20381.8} C_VEL
LIN {X 0,Y 450.116,Z 441.728,A -85,B 0,C 180,E1 20379.938,E2 20379.938} C_VEL
LIN {X 0,Y 447.644,Z 425.997,A -85,B 0,C 180,E1 20378.059,E2 20378.059} C_VEL
LIN {X 0,Y 447.095,Z 408.118,A -85,B 0,C 180,E1 20376.105,E2 20376.105} C_VEL
LIN {X 0,Y 448.853,Z 386.752,A -85,B 0,C 180,E1 20373.995,E2 20373.995} C_VEL
LIN {X 0,Y 454.535,Z 347.141,A -85,B 0,C 180,E1 20370.247,E2 20370.247} C_VEL
LIN {X 0,Y 454.905,Z 343.7,A -85,B 0,C 180,E1 20369.893,E2 20369.893} C_VEL
LIN {X 0,Y 443.045,Z 348.381,A -85,B 0,C 180,E1 20368.583,E2 20368.583} C_VEL
LIN {X 0,Y 438.307,Z 350.238,A -85,B 0,C 180,E1 20368.029,E2 20368.029} C_VEL
LIN {X 0,Y 434.36,Z 351.852,A -85,B 0,C 180,E1 20367.56,E2 20367.56} C_VEL
LIN {X 0,Y 433.252,Z 352.208,A -85,B 0,C 180,E1 20367.413,E2 20367.413} C_VEL
LIN {X 0,Y 430.126,Z 353.916,A -85,B 0,C 180,E1 20367.086,E2 20367.086} C_VEL
LIN {X 0,Y 427.841,Z 354.159,A -85,B 0,C 180,E1 20366.679,E2 20366.679} C_VEL
LIN {X 0,Y 427.248,Z 397.912,A -85,B 0,C 180,E1 20363.443,E2 20363.443} C_VEL
LIN {X 0,Y 426.215,Z 447.777,A -85,B 0,C 180,E1 20359.672,E2 20359.672} C_VEL
LIN {X 0,Y 425.043,Z 494.402,A -85,B 0,C 180,E1 20356.045,E2 20356.045} C_VEL
LIN {X 0,Y 424.481,Z 505.975,A -85,B 0,C 180,E1 20355.156,E2 20355.156} C_VEL
LIN {X 0,Y 423.098,Z 514.636,A -85,B 0,C 180,E1 20354.59,E2 20354.59} C_VEL
LIN {X 0,Y 421.254,Z 613.888,A -85,B 0,C 180,E1 20352.549,E2 20352.549} C_VEL
LIN {X 0,Y 421.355,Z 631.537,A -85,B 0,C 180,E1 20352.106,E2 20352.106} C_VEL
LIN {X 0,Y 421.292,Z 645.785,A -85,B 0,C 180,E1 20351.499,E2 20351.499} C_VEL
LIN {X 0,Y 421.035,Z 659.348,A -85,B 0,C 180,E1 20350.674,E2 20350.674} C_VEL
LIN {X 0,Y 420.669,Z 671.948,A -85,B 0,C 180,E1 20349.646,E2 20349.646} C_VEL
LIN {X 0,Y 420.172,Z 684.095,A -85,B 0,C 180,E1 20348.346,E2 20348.346} C_VEL
LIN {X 0,Y 419.616,Z 694.893,A -85,B 0,C 180,E1 20346.842,E2 20346.842} C_VEL
LIN {X 0,Y 419.08,Z 703.958,A -85,B 0,C 180,E1 20345.201,E2 20345.201} C_VEL
LIN {X 0,Y 418.629,Z 710.889,A -85,B 0,C 180,E1 20343.56,E2 20343.56} C_VEL
LIN {X 0,Y 418.245,Z 716.448,A -85,B 0,C 180,E1 20341.78,E2 20341.78} C_VEL
LIN {X 0,Y 417.934,Z 720.439,A -85,B 0,C 180,E1 20339.862,E2 20339.862} C_VEL
LIN {X 0,Y 417.737,Z 722.617,A -85,B 0,C 180,E1 20337.942,E2 20337.942} C_VEL
LIN {X 0,Y 417.615,Z 723.089,A -85,B 0,C 180,E1 20336.018,E2 20336.018} C_VEL
LIN {X 0,Y 417.581,Z 721.665,A -85,B 0,C 180,E1 20333.952,E2 20333.952} C_VEL
LIN {X 0,Y 417.628,Z 718.531,A -85,B 0,C 180,E1 20332.018,E2 20332.018} C_VEL
LIN {X 0,Y 417.778,Z 713.974,A -85,B 0,C 180,E1 20330.216,E2 20330.216} C_VEL
LIN {X 0,Y 418.055,Z 707.01,A -85,B 0,C 180,E1 20328.27,E2 20328.27} C_VEL
LIN {X 0,Y 418.451,Z 698.277,A -85,B 0,C 180,E1 20326.457,E2 20326.457} C_VEL
LIN {X 0,Y 418.921,Z 687.714,A -85,B 0,C 180,E1 20324.778,E2 20324.778} C_VEL
LIN {X 0,Y 419.424,Z 675.743,A -85,B 0,C 180,E1 20323.306,E2 20323.306} C_VEL
LIN {X 0,Y 419.898,Z 662.382,A -85,B 0,C 180,E1 20322.039,E2 20322.039} C_VEL
LIN {X 0,Y 420.297,Z 648.585,A -85,B 0,C 180,E1 20321.051,E2 20321.051} C_VEL
LIN {X 0,Y 420.55,Z 633.926,A -85,B 0,C 180,E1 20320.288,E2 20320.288} C_VEL
LIN {X 0,Y 420.654,Z 619.035,A -85,B 0,C 180,E1 20319.775,E2 20319.775} C_VEL
LIN {X 0,Y 422.267,Z 503.799,A -85,B 0,C 180,E1 20317.517,E2 20317.517} C_VEL
LIN {X 0,Y 422.905,Z 492.255,A -85,B 0,C 180,E1 20316.596,E2 20316.596} C_VEL
LIN {X 0,Y 424.432,Z 443.58,A -85,B 0,C 180,E1 20312.639,E2 20312.639} C_VEL
LIN {X 0,Y 425.938,Z 396.83,A -85,B 0,C 180,E1 20308.827,E2 20308.827} C_VEL
LIN {X 0,Y 427.403,Z 351.465,A -85,B 0,C 180,E1 20305.111,E2 20305.111} C_VEL
LIN {X 0,Y 428.775,Z 306.059,A -85,B 0,C 180,E1 20301.37,E2 20301.37} C_VEL
LIN {X 0,Y 430.466,Z 305.897,A -85,B 0,C 180,E1 20300.989,E2 20300.989} C_VEL
LIN {X 0,Y 433.981,Z 303.938,A -85,B 0,C 180,E1 20300.514,E2 20300.514} C_VEL
LIN {X 0,Y 438.237,Z 302.589,A -85,B 0,C 180,E1 20299.783,E2 20299.783} C_VEL
LIN {X 0,Y 439.205,Z 302.694,A -85,B 0,C 180,E1 20299.547,E2 20299.547} C_VEL
LIN {X 0,Y 444.707,Z 315.105,A -85,B 0,C 180,E1 20296.35,E2 20296.35} C_VEL
LIN {X 0,Y 450.228,Z 328.895,A -85,B 0,C 180,E1 20293.245,E2 20293.245} C_VEL
LIN {X 0,Y 450.441,Z 329.731,A -85,B 0,C 180,E1 20293.088,E2 20293.088} C_VEL
LIN {X 0,Y 449.388,Z 337.509,A -85,B 0,C 180,E1 20292.223,E2 20292.223} C_VEL
LIN {X 0,Y 449.725,Z 340.256,A -85,B 0,C 180,E1 20292.124,E2 20292.124} C_VEL
LIN {X 0,Y 447.069,Z 418.843,A -85,B 0,C 180,E1 20290.694,E2 20290.694} C_VEL
LIN {X 0,Y 445.359,Z 455.61,A -85,B 0,C 180,E1 20289.952,E2 20289.952} C_VEL
LIN {X 0,Y 444.218,Z 463.269,A -85,B 0,C 180,E1 20289.874,E2 20289.874} C_VEL
LIN {X 0,Y 438.36,Z 483.688,A -85,B 0,C 180,E1 20289.963,E2 20289.963} C_VEL
LIN {X 0,Y 437.435,Z 490.248,A -85,B 0,C 180,E1 20289.878,E2 20289.878} C_VEL
LIN {X 0,Y 432.263,Z 575.818,A -85,B 0,C 180,E1 20287.805,E2 20287.805} C_VEL
LIN {X 0,Y 430.947,Z 596.445,A -85,B 0,C 180,E1 20287.108,E2 20287.108} C_VEL
LIN {X 0,Y 429.23,Z 616.25,A -85,B 0,C 180,E1 20286.194,E2 20286.194} C_VEL
LIN {X 0,Y 427.191,Z 635.175,A -85,B 0,C 180,E1 20285.072,E2 20285.072} C_VEL
LIN {X 0,Y 424.809,Z 654.209,A -85,B 0,C 180,E1 20283.662,E2 20283.662} C_VEL
LIN {X 0,Y 422.288,Z 672.211,A -85,B 0,C 180,E1 20282.031,E2 20282.031} C_VEL
LIN {X 0,Y 419.662,Z 689.54,A -85,B 0,C 180,E1 20280.132,E2 20280.132} C_VEL
LIN {X 0,Y 417.142,Z 705.565,A -85,B 0,C 180,E1 20278.021,E2 20278.021} C_VEL
LIN {X 0,Y 414.819,Z 720.213,A -85,B 0,C 180,E1 20275.713,E2 20275.713} C_VEL
LIN {X 0,Y 412.82,Z 733.252,A -85,B 0,C 180,E1 20273.253,E2 20273.253} C_VEL
LIN {X 0,Y 411.187,Z 744.731,A -85,B 0,C 180,E1 20270.646,E2 20270.646} C_VEL
LIN {X 0,Y 409.948,Z 754.631,A -85,B 0,C 180,E1 20267.898,E2 20267.898} C_VEL
LIN {X 0,Y 409.081,Z 762.696,A -85,B 0,C 180,E1 20265.104,E2 20265.104} C_VEL
LIN {X 0,Y 408.557,Z 769.233,A -85,B 0,C 180,E1 20262.15,E2 20262.15} C_VEL
LIN {X 0,Y 408.289,Z 773.758,A -85,B 0,C 180,E1 20259.278,E2 20259.278} C_VEL
LIN {X 0,Y 408.173,Z 776.518,A -85,B 0,C 180,E1 20256.47,E2 20256.47} C_VEL
LIN {X 0,Y 408.138,Z 777.694,A -85,B 0,C 180,E1 20253.652,E2 20253.652} C_VEL
LIN {X 0,Y 408.142,Z 777.282,A -85,B 0,C 180,E1 20250.842,E2 20250.842} C_VEL
LIN {X 0,Y 408.206,Z 775.442,A -85,B 0,C 180,E1 20248.175,E2 20248.175} C_VEL
LIN {X 0,Y 408.373,Z 771.904,A -85,B 0,C 180,E1 20245.366,E2 20245.366} C_VEL
LIN {X 0,Y 408.718,Z 766.64,A -85,B 0,C 180,E1 20242.55,E2 20242.55} C_VEL
LIN {X 0,Y 409.292,Z 759.972,A -85,B 0,C 180,E1 20239.87,E2 20239.87} C_VEL
LIN {X 0,Y 410.245,Z 751.378,A -85,B 0,C 180,E1 20237.136,E2 20237.136} C_VEL
LIN {X 0,Y 411.547,Z 741.152,A -85,B 0,C 180,E1 20234.499,E2 20234.499} C_VEL
LIN {X 0,Y 413.237,Z 729.199,A -85,B 0,C 180,E1 20231.958,E2 20231.958} C_VEL
LIN {X 0,Y 415.259,Z 715.681,A -85,B 0,C 180,E1 20229.566,E2 20229.566} C_VEL
LIN {X 0,Y 417.566,Z 700.525,A -85,B 0,C 180,E1 20227.324,E2 20227.324} C_VEL
LIN {X 0,Y 420.028,Z 684.183,A -85,B 0,C 180,E1 20225.306,E2 20225.306} C_VEL
LIN {X 0,Y 422.519,Z 666.7,A -85,B 0,C 180,E1 20223.508,E2 20223.508} C_VEL
LIN {X 0,Y 424.841,Z 648.938,A -85,B 0,C 180,E1 20221.997,E2 20221.997} C_VEL
LIN {X 0,Y 426.998,Z 630.347,A -85,B 0,C 180,E1 20220.699,E2 20220.699} C_VEL
LIN {X 0,Y 428.966,Z 610.343,A -85,B 0,C 180,E1 20219.59,E2 20219.59} C_VEL
LIN {X 0,Y 430.516,Z 590.201,A -85,B 0,C 180,E1 20218.737,E2 20218.737} C_VEL
LIN {X 0,Y 431.84,Z 567.36,A -85,B 0,C 180,E1 20218.053,E2 20218.053} C_VEL
LIN {X 0,Y 436.854,Z 479.876,A -85,B 0,C 180,E1 20215.991,E2 20215.991} C_VEL
LIN {X 0,Y 440.367,Z 405.637,A -85,B 0,C 180,E1 20214.466,E2 20214.466} C_VEL
LIN {X 0,Y 442.589,Z 336.81,A -85,B 0,C 180,E1 20213.225,E2 20213.225} C_VEL
LIN {X 0,Y 443.585,Z 330.481,A -85,B 0,C 180,E1 20212.654,E2 20212.654} C_VEL
LIN {X 0,Y 436.427,Z 313.989,A -85,B 0,C 180,E1 20209.519,E2 20209.519} C_VEL
LIN {X 0,Y 429.586,Z 299.367,A -85,B 0,C 180,E1 20206.374,E2 20206.374} C_VEL
LIN {X 0,Y 424.574,Z 289.64,A -85,B 0,C 180,E1 20204.005,E2 20204.005} C_VEL
LIN {X 0,Y 420.401,Z 281.585,A -85,B 0,C 180,E1 20201.89,E2 20201.89} C_VEL
LIN {X 0,Y 417.623,Z 276.588,A -85,B 0,C 180,E1 20200.453,E2 20200.453} C_VEL
LIN {X 0,Y 415.215,Z 272.078,A -85,B 0,C 180,E1 20199.118,E2 20199.118} C_VEL
LIN {X 0,Y 412.996,Z 268.637,A -85,B 0,C 180,E1 20197.948,E2 20197.948} C_VEL
LIN {X 0,Y 412.376,Z 266.967,A -85,B 0,C 180,E1 20197.488,E2 20197.488} C_VEL
LIN {X 0,Y 410.118,Z 264.095,A -85,B 0,C 180,E1 20196.33,E2 20196.33} C_VEL
LIN {X 0,Y 409.432,Z 261.718,A -85,B 0,C 180,E1 20195.614,E2 20195.614} C_VEL
LIN {X 0,Y 418.395,Z 287.594,A -85,B 0,C 180,E1 20192.479,E2 20192.479} C_VEL
LIN {X 0,Y 422.158,Z 299.72,A -85,B 0,C 180,E1 20191.087,E2 20191.087} C_VEL
LIN {X 0,Y 420.841,Z 341.552,A -85,B 0,C 180,E1 20187.37,E2 20187.37} C_VEL
LIN {X 0,Y 419.378,Z 384.066,A -85,B 0,C 180,E1 20183.612,E2 20183.612} C_VEL
LIN {X 0,Y 417.765,Z 429.063,A -85,B 0,C 180,E1 20179.65,E2 20179.65} C_VEL
LIN {X 0,Y 416.898,Z 455.502,A -85,B 0,C 180,E1 20177.355,E2 20177.355} C_VEL
LIN {X 0,Y 414.346,Z 599.526,A -85,B 0,C 180,E1 20174.437,E2 20174.437} C_VEL
LIN {X 0,Y 414.122,Z 616.826,A -85,B 0,C 180,E1 20173.83,E2 20173.83} C_VEL
LIN {X 0,Y 413.69,Z 632.953,A -85,B 0,C 180,E1 20172.99,E2 20172.99} C_VEL
LIN {X 0,Y 413.141,Z 648.031,A -85,B 0,C 180,E1 20171.943,E2 20171.943} C_VEL
LIN {X 0,Y 412.495,Z 662.811,A -85,B 0,C 180,E1 20170.616,E2 20170.616} C_VEL
LIN {X 0,Y 411.806,Z 676.239,A -85,B 0,C 180,E1 20169.081,E2 20169.081} C_VEL
LIN {X 0,Y 411.218,Z 687.119,A -85,B 0,C 180,E1 20167.545,E2 20167.545} C_VEL
LIN {X 0,Y 410.656,Z 697.425,A -85,B 0,C 180,E1 20165.73,E2 20165.73} C_VEL
LIN {X 0,Y 410.255,Z 705.681,A -85,B 0,C 180,E1 20163.913,E2 20163.913} C_VEL
LIN {X 0,Y 409.939,Z 713,A -85,B 0,C 180,E1 20161.818,E2 20161.818} C_VEL
LIN {X 0,Y 409.764,Z 718.373,A -85,B 0,C 180,E1 20159.721,E2 20159.721} C_VEL
LIN {X 0,Y 409.7,Z 722.148,A -85,B 0,C 180,E1 20157.483,E2 20157.483} C_VEL
LIN {X 0,Y 409.747,Z 723.92,A -85,B 0,C 180,E1 20155.382,E2 20155.382} C_VEL
LIN {X 0,Y 409.895,Z 724.018,A -85,B 0,C 180,E1 20153.136,E2 20153.136} C_VEL
LIN {X 0,Y 410.121,Z 722.285,A -85,B 0,C 180,E1 20151.024,E2 20151.024} C_VEL
LIN {X 0,Y 410.48,Z 718.814,A -85,B 0,C 180,E1 20148.906,E2 20148.906} C_VEL
LIN {X 0,Y 410.895,Z 713.764,A -85,B 0,C 180,E1 20146.921,E2 20146.921} C_VEL
LIN {X 0,Y 411.466,Z 706.801,A -85,B 0,C 180,E1 20144.93,E2 20144.93} C_VEL
LIN {X 0,Y 412.111,Z 698.158,A -85,B 0,C 180,E1 20143.074,E2 20143.074} C_VEL
LIN {X 0,Y 412.818,Z 687.955,A -85,B 0,C 180,E1 20141.355,E2 20141.355} C_VEL
LIN {X 0,Y 413.54,Z 676.017,A -85,B 0,C 180,E1 20139.773,E2 20139.773} C_VEL
LIN {X 0,Y 414.15,Z 663.569,A -85,B 0,C 180,E1 20138.472,E2 20138.472} C_VEL
LIN {X 0,Y 414.672,Z 649.42,A -85,B 0,C 180,E1 20137.308,E2 20137.308} C_VEL
LIN {X 0,Y 415.059,Z 633.4,A -85,B 0,C 180,E1 20136.316,E2 20136.316} C_VEL
LIN {X 0,Y 415.225,Z 617.362,A -85,B 0,C 180,E1 20135.614,E2 20135.614} C_VEL
LIN {X 0,Y 415.168,Z 600.342,A -85,B 0,C 180,E1 20135.136,E2 20135.136} C_VEL
LIN {X 0,Y 416.527,Z 533.485,A -85,B 0,C 180,E1 20133.689,E2 20133.689} C_VEL
LIN {X 0,Y 418.598,Z 471.539,A -85,B 0,C 180,E1 20132.24,E2 20132.24} C_VEL
LIN {X 0,Y 420.91,Z 459.418,A -85,B 0,C 180,E1 20131.403,E2 20131.403} C_VEL
LIN {X 0,Y 422.14,Z 416.942,A -85,B 0,C 180,E1 20127.877,E2 20127.877} C_VEL
LIN {X 0,Y 422.807,Z 394.072,A -85,B 0,C 180,E1 20125.995,E2 20125.995} C_VEL
LIN {X 0,Y 425.242,Z 394.221,A -85,B 0,C 180,E1 20125.647,E2 20125.647} C_VEL
LIN {X 0,Y 427.878,Z 393.104,A -85,B 0,C 180,E1 20125.401,E2 20125.401} C_VEL
LIN {X 0,Y 429.568,Z 392.341,A -85,B 0,C 180,E1 20125.25,E2 20125.25} C_VEL
LIN {X 0,Y 433.815,Z 391.057,A -85,B 0,C 180,E1 20124.817,E2 20124.817} C_VEL
LIN {X 0,Y 436.364,Z 390.198,A -85,B 0,C 180,E1 20124.57,E2 20124.57} C_VEL
LIN {X 0,Y 445.349,Z 387.337,A -85,B 0,C 180,E1 20123.716,E2 20123.716} C_VEL
LIN {X 0,Y 447.47,Z 404.638,A -85,B 0,C 180,E1 20121.924,E2 20121.924} C_VEL
LIN {X 0,Y 451.444,Z 420.531,A -85,B 0,C 180,E1 20120.12,E2 20120.12} C_VEL
LIN {X 0,Y 456.826,Z 433.943,A -85,B 0,C 180,E1 20118.458,E2 20118.458} C_VEL
LIN {X 0,Y 464.277,Z 446.943,A -85,B 0,C 180,E1 20116.712,E2 20116.712} C_VEL
LIN {X 0,Y 473.622,Z 458.673,A -85,B 0,C 180,E1 20114.992,E2 20114.992} C_VEL
LIN {X 0,Y 480.753,Z 465.824,A -85,B 0,C 180,E1 20113.875,E2 20113.875} C_VEL
LIN {X 0,Y 469.156,Z 485.685,A -85,B 0,C 180,E1 20113.334,E2 20113.334} C_VEL
LIN {X 0,Y 460.658,Z 503.011,A -85,B 0,C 180,E1 20112.71,E2 20112.71} C_VEL
LIN {X 0,Y 449.861,Z 524.784,A -85,B 0,C 180,E1 20111.905,E2 20111.905} C_VEL
LIN {X 0,Y 442.793,Z 542.677,A -85,B 0,C 180,E1 20111.114,E2 20111.114} C_VEL
LIN {X 0,Y 440.481,Z 561.398,A -85,B 0,C 180,E1 20110.961,E2 20110.961} C_VEL
LIN {X 0,Y 439.495,Z 577.933,A -85,B 0,C 180,E1 20110.715,E2 20110.715} C_VEL
LIN {X 0,Y 438.035,Z 604.235,A -85,B 0,C 180,E1 20110.115,E2 20110.115} C_VEL
LIN {X 0,Y 435.727,Z 630.019,A -85,B 0,C 180,E1 20109.297,E2 20109.297} C_VEL
LIN {X 0,Y 433.312,Z 653.92,A -85,B 0,C 180,E1 20108.284,E2 20108.284} C_VEL
LIN {X 0,Y 430.667,Z 676.912,A -85,B 0,C 180,E1 20107.047,E2 20107.047} C_VEL
LIN {X 0,Y 427.903,Z 698.995,A -85,B 0,C 180,E1 20105.579,E2 20105.579} C_VEL
LIN {X 0,Y 425.049,Z 720.145,A -85,B 0,C 180,E1 20103.884,E2 20103.884} C_VEL
LIN {X 0,Y 422.31,Z 739.327,A -85,B 0,C 180,E1 20102.049,E2 20102.049} C_VEL
LIN {X 0,Y 419.507,Z 757.446,A -85,B 0,C 180,E1 20099.956,E2 20099.956} C_VEL
LIN {X 0,Y 417.069,Z 772.589,A -85,B 0,C 180,E1 20097.871,E2 20097.871} C_VEL
LIN {X 0,Y 414.638,Z 787.632,A -85,B 0,C 180,E1 20095.419,E2 20095.419} C_VEL
LIN {X 0,Y 412.554,Z 801.035,A -85,B 0,C 180,E1 20092.816,E2 20092.816} C_VEL
LIN {X 0,Y 410.886,Z 813.023,A -85,B 0,C 180,E1 20090.067,E2 20090.067} C_VEL
LIN {X 0,Y 409.572,Z 824.014,A -85,B 0,C 180,E1 20087.035,E2 20087.035} C_VEL
LIN {X 0,Y 408.694,Z 833.273,A -85,B 0,C 180,E1 20083.872,E2 20083.872} C_VEL
LIN {X 0,Y 408.243,Z 840.213,A -85,B 0,C 180,E1 20080.853,E2 20080.853} C_VEL
LIN {X 0,Y 408.035,Z 845.361,A -85,B 0,C 180,E1 20077.887,E2 20077.887} C_VEL
LIN {X 0,Y 407.973,Z 848.969,A -85,B 0,C 180,E1 20074.78,E2 20074.78} C_VEL
LIN {X 0,Y 407.965,Z 850.699,A -85,B 0,C 180,E1 20071.966,E2 20071.966} C_VEL
LIN {X 0,Y 407.97,Z 850.97,A -85,B 0,C 180,E1 20069.017,E2 20069.017} C_VEL
LIN {X 0,Y 407.966,Z 849.622,A -85,B 0,C 180,E1 20066.065,E2 20066.065} C_VEL
LIN {X 0,Y 408.005,Z 846.695,A -85,B 0,C 180,E1 20063.103,E2 20063.103} C_VEL
LIN {X 0,Y 408.16,Z 841.808,A -85,B 0,C 180,E1 20059.984,E2 20059.984} C_VEL
LIN {X 0,Y 408.535,Z 835.384,A -85,B 0,C 180,E1 20056.987,E2 20056.987} C_VEL
LIN {X 0,Y 409.237,Z 827.131,A -85,B 0,C 180,E1 20053.973,E2 20053.973} C_VEL
LIN {X 0,Y 410.446,Z 816.317,A -85,B 0,C 180,E1 20050.8,E2 20050.8} C_VEL
LIN {X 0,Y 412.054,Z 804.309,A -85,B 0,C 180,E1 20047.907,E2 20047.907} C_VEL
LIN {X 0,Y 414.058,Z 791.012,A -85,B 0,C 180,E1 20045.224,E2 20045.224} C_VEL
LIN {X 0,Y 416.437,Z 776.211,A -85,B 0,C 180,E1 20042.704,E2 20042.704} C_VEL
LIN {X 0,Y 419.137,Z 759.51,A -85,B 0,C 180,E1 20040.33,E2 20040.33} C_VEL
LIN {X 0,Y 421.737,Z 742.775,A -85,B 0,C 180,E1 20038.333,E2 20038.333} C_VEL
LIN {X 0,Y 424.276,Z 725.613,A -85,B 0,C 180,E1 20036.614,E2 20036.614} C_VEL
LIN {X 0,Y 427.01,Z 706.031,A -85,B 0,C 180,E1 20034.933,E2 20034.933} C_VEL
LIN {X 0,Y 429.755,Z 685.098,A -85,B 0,C 180,E1 20033.444,E2 20033.444} C_VEL
LIN {X 0,Y 432.467,Z 662.936,A -85,B 0,C 180,E1 20032.132,E2 20032.132} C_VEL
LIN {X 0,Y 435.083,Z 639.104,A -85,B 0,C 180,E1 20031.005,E2 20031.005} C_VEL
LIN {X 0,Y 437.513,Z 614.286,A -85,B 0,C 180,E1 20030.115,E2 20030.115} C_VEL
LIN {X 0,Y 439.392,Z 589.04,A -85,B 0,C 180,E1 20029.448,E2 20029.448} C_VEL
LIN {X 0,Y 440.579,Z 566.271,A -85,B 0,C 180,E1 20029.023,E2 20029.023} C_VEL
LIN {X 0,Y 443.246,Z 545.456,A -85,B 0,C 180,E1 20028.873,E2 20028.873} C_VEL
LIN {X 0,Y 443.84,Z 542.158,A -85,B 0,C 180,E1 20028.867,E2 20028.867} C_VEL
LIN {X 0,Y 452.989,Z 523.9,A -85,B 0,C 180,E1 20027.94,E2 20027.94} C_VEL
LIN {X 0,Y 462.342,Z 508.717,A -85,B 0,C 180,E1 20027.331,E2 20027.331} C_VEL
LIN {X 0,Y 471.044,Z 494.392,A -85,B 0,C 180,E1 20026.766,E2 20026.766} C_VEL
LIN {X 0,Y 461.133,Z 483.504,A -85,B 0,C 180,E1 20024.979,E2 20024.979} C_VEL
LIN {X 0,Y 453.223,Z 471.496,A -85,B 0,C 180,E1 20023.148,E2 20023.148} C_VEL
LIN {X 0,Y 447.036,Z 457.682,A -85,B 0,C 180,E1 20021.2,E2 20021.2} C_VEL
LIN {X 0,Y 443.129,Z 443.458,A -85,B 0,C 180,E1 20019.348,E2 20019.348} C_VEL
LIN {X 0,Y 440.927,Z 426.738,A -85,B 0,C 180,E1 20017.343,E2 20017.343} C_VEL
LIN {X 0,Y 440.804,Z 408.411,A -85,B 0,C 180,E1 20015.338,E2 20015.338} C_VEL
LIN {X 0,Y 443.141,Z 385.7,A -85,B 0,C 180,E1 20013.094,E2 20013.094} C_VEL
LIN {X 0,Y 448.228,Z 352.176,A -85,B 0,C 180,E1 20009.886,E2 20009.886} C_VEL
LIN {X 0,Y 435.756,Z 357.263,A -85,B 0,C 180,E1 20008.506,E2 20008.506} C_VEL
LIN {X 0,Y 431.465,Z 359.004,A -85,B 0,C 180,E1 20008.003,E2 20008.003} C_VEL
LIN {X 0,Y 427.198,Z 360.795,A -85,B 0,C 180,E1 20007.494,E2 20007.494} C_VEL
LIN {X 0,Y 426.267,Z 361.108,A -85,B 0,C 180,E1 20007.37,E2 20007.37} C_VEL
LIN {X 0,Y 422.844,Z 362.94,A -85,B 0,C 180,E1 20007,E2 20007} C_VEL
LIN {X 0,Y 420.83,Z 363.221,A -85,B 0,C 180,E1 20006.625,E2 20006.625} C_VEL
LIN {X 0,Y 419.989,Z 408.954,A -85,B 0,C 180,E1 20003.181,E2 20003.181} C_VEL
LIN {X 0,Y 418.995,Z 451.277,A -85,B 0,C 180,E1 19999.952,E2 19999.952} C_VEL
LIN {X 0,Y 417.655,Z 500.043,A -85,B 0,C 180,E1 19996.123,E2 19996.123} C_VEL
LIN {X 0,Y 417.149,Z 507.251,A -85,B 0,C 180,E1 19995.572,E2 19995.572} C_VEL
LIN {X 0,Y 415.666,Z 516.432,A -85,B 0,C 180,E1 19994.972,E2 19994.972} C_VEL
LIN {X 0,Y 413.666,Z 612.337,A -85,B 0,C 180,E1 19992.934,E2 19992.934} C_VEL
LIN {X 0,Y 413.769,Z 631.728,A -85,B 0,C 180,E1 19992.459,E2 19992.459} C_VEL
LIN {X 0,Y 413.716,Z 646.147,A -85,B 0,C 180,E1 19991.854,E2 19991.854} C_VEL
LIN {X 0,Y 413.448,Z 660.024,A -85,B 0,C 180,E1 19991.014,E2 19991.014} C_VEL
LIN {X 0,Y 413.025,Z 673.519,A -85,B 0,C 180,E1 19989.897,E2 19989.897} C_VEL
LIN {X 0,Y 412.497,Z 685.679,A -85,B 0,C 180,E1 19988.573,E2 19988.573} C_VEL
LIN {X 0,Y 411.929,Z 696.035,A -85,B 0,C 180,E1 19987.11,E2 19987.11} C_VEL
LIN {X 0,Y 411.396,Z 704.511,A -85,B 0,C 180,E1 19985.578,E2 19985.578} C_VEL
LIN {X 0,Y 410.892,Z 711.736,A -85,B 0,C 180,E1 19983.889,E2 19983.889} C_VEL
LIN {X 0,Y 410.434,Z 717.748,A -85,B 0,C 180,E1 19981.954,E2 19981.954} C_VEL
LIN {X 0,Y 410.092,Z 721.779,A -85,B 0,C 180,E1 19979.999,E2 19979.999} C_VEL
LIN {X 0,Y 409.871,Z 723.98,A -85,B 0,C 180,E1 19978.042,E2 19978.042} C_VEL
LIN {X 0,Y 409.733,Z 724.451,A -85,B 0,C 180,E1 19976.082,E2 19976.082} C_VEL
LIN {X 0,Y 409.688,Z 723.011,A -85,B 0,C 180,E1 19973.976,E2 19973.976} C_VEL
LIN {X 0,Y 409.733,Z 719.859,A -85,B 0,C 180,E1 19972.004,E2 19972.004} C_VEL
LIN {X 0,Y 409.886,Z 715.269,A -85,B 0,C 180,E1 19970.168,E2 19970.168} C_VEL
LIN {X 0,Y 410.151,Z 708.844,A -85,B 0,C 180,E1 19968.326,E2 19968.326} C_VEL
LIN {X 0,Y 410.549,Z 700.24,A -85,B 0,C 180,E1 19966.479,E2 19966.479} C_VEL
LIN {X 0,Y 410.985,Z 690.805,A -85,B 0,C 180,E1 19964.911,E2 19964.911} C_VEL
LIN {X 0,Y 411.467,Z 679.96,A -85,B 0,C 180,E1 19963.482,E2 19963.482} C_VEL
LIN {X 0,Y 411.957,Z 667.499,A -85,B 0,C 180,E1 19962.192,E2 19962.192} C_VEL
LIN {X 0,Y 412.394,Z 653.925,A -85,B 0,C 180,E1 19961.114,E2 19961.114} C_VEL
LIN {X 0,Y 412.728,Z 638.584,A -85,B 0,C 180,E1 19960.223,E2 19960.223} C_VEL
LIN {X 0,Y 412.883,Z 622.383,A -85,B 0,C 180,E1 19959.6,E2 19959.6} C_VEL
LIN {X 0,Y 413.188,Z 581.357,A -85,B 0,C 180,E1 19958.765,E2 19958.765} C_VEL
LIN {X 0,Y 414.575,Z 504.884,A -85,B 0,C 180,E1 19957.226,E2 19957.226} C_VEL
LIN {X 0,Y 415.2,Z 496.028,A -85,B 0,C 180,E1 19956.52,E2 19956.52} C_VEL
LIN {X 0,Y 416.814,Z 446.441,A -85,B 0,C 180,E1 19952.46,E2 19952.46} C_VEL
LIN {X 0,Y 418.405,Z 399.551,A -85,B 0,C 180,E1 19948.603,E2 19948.603} C_VEL
LIN {X 0,Y 419.958,Z 353.658,A -85,B 0,C 180,E1 19944.818,E2 19944.818} C_VEL
LIN {X 0,Y 421.218,Z 314.853,A -85,B 0,C 180,E1 19941.586,E2 19941.586} C_VEL
LIN {X 0,Y 422.878,Z 314.695,A -85,B 0,C 180,E1 19941.202,E2 19941.202} C_VEL
LIN {X 0,Y 426.065,Z 312.933,A -85,B 0,C 180,E1 19940.753,E2 19940.753} C_VEL
LIN {X 0,Y 430.176,Z 311.203,A -85,B 0,C 180,E1 19940.095,E2 19940.095} C_VEL
LIN {X 0,Y 432.261,Z 310.118,A -85,B 0,C 180,E1 19939.807,E2 19939.807} C_VEL
LIN {X 0,Y 434.282,Z 309.43,A -85,B 0,C 180,E1 19939.472,E2 19939.472} C_VEL
LIN {X 0,Y 439.518,Z 321.594,A -85,B 0,C 180,E1 19936.338,E2 19936.338} C_VEL
LIN {X 0,Y 444.397,Z 333.954,A -85,B 0,C 180,E1 19933.532,E2 19933.532} C_VEL
LIN {X 0,Y 443.598,Z 339.864,A -85,B 0,C 180,E1 19932.876,E2 19932.876} C_VEL
LIN {X 0,Y 443.816,Z 342.702,A -85,B 0,C 180,E1 19932.787,E2 19932.787} C_VEL
LIN {X 0,Y 441.071,Z 419.92,A -85,B 0,C 180,E1 19931.366,E2 19931.366} C_VEL
LIN {X 0,Y 437.435,Z 490.248,A -85,B 0,C 180,E1 19929.878,E2 19929.878} C_VEL
LIN {X 0,Y 436.248,Z 497.89,A -85,B 0,C 180,E1 19929.787,E2 19929.787} C_VEL
LIN {X 0,Y 430.204,Z 518.263,A -85,B 0,C 180,E1 19929.845,E2 19929.845} C_VEL
LIN {X 0,Y 429.211,Z 524.812,A -85,B 0,C 180,E1 19929.751,E2 19929.751} C_VEL
LIN {X 0,Y 425.546,Z 581.435,A -85,B 0,C 180,E1 19928.283,E2 19928.283} C_VEL
LIN {X 0,Y 424.02,Z 602.124,A -85,B 0,C 180,E1 19927.515,E2 19927.515} C_VEL
LIN {X 0,Y 422.033,Z 622.524,A -85,B 0,C 180,E1 19926.489,E2 19926.489} C_VEL
LIN {X 0,Y 419.8,Z 641.426,A -85,B 0,C 180,E1 19925.273,E2 19925.273} C_VEL
LIN {X 0,Y 417.214,Z 660.175,A -85,B 0,C 180,E1 19923.779,E2 19923.779} C_VEL
LIN {X 0,Y 414.536,Z 677.969,A -85,B 0,C 180,E1 19922.049,E2 19922.049} C_VEL
LIN {X 0,Y 411.809,Z 694.685,A -85,B 0,C 180,E1 19920.091,E2 19920.091} C_VEL
LIN {X 0,Y 409.185,Z 710.284,A -85,B 0,C 180,E1 19917.901,E2 19917.901} C_VEL
LIN {X 0,Y 406.875,Z 724.052,A -85,B 0,C 180,E1 19915.594,E2 19915.594} C_VEL
LIN {X 0,Y 404.87,Z 736.42,A -85,B 0,C 180,E1 19913.121,E2 19913.121} C_VEL
LIN {X 0,Y 403.157,Z 747.821,A -85,B 0,C 180,E1 19910.368,E2 19910.368} C_VEL
LIN {X 0,Y 401.893,Z 757.392,A -85,B 0,C 180,E1 19907.52,E2 19907.52} C_VEL
LIN {X 0,Y 401.036,Z 765.197,A -85,B 0,C 180,E1 19904.585,E2 19904.585} C_VEL
LIN {X 0,Y 400.546,Z 771.09,A -85,B 0,C 180,E1 19901.666,E2 19901.666} C_VEL
LIN {X 0,Y 400.304,Z 775.215,A -85,B 0,C 180,E1 19898.764,E2 19898.764} C_VEL
LIN {X 0,Y 400.205,Z 777.608,A -85,B 0,C 180,E1 19896.023,E2 19896.023} C_VEL
LIN {X 0,Y 400.172,Z 778.49,A -85,B 0,C 180,E1 19893.151,E2 19893.151} C_VEL
LIN {X 0,Y 400.178,Z 777.818,A -85,B 0,C 180,E1 19890.43,E2 19890.43} C_VEL
LIN {X 0,Y 400.269,Z 775.579,A -85,B 0,C 180,E1 19887.566,E2 19887.566} C_VEL
LIN {X 0,Y 400.483,Z 771.721,A -85,B 0,C 180,E1 19884.7,E2 19884.7} C_VEL
LIN {X 0,Y 400.883,Z 766.485,A -85,B 0,C 180,E1 19881.966,E2 19881.966} C_VEL
LIN {X 0,Y 401.619,Z 759.2,A -85,B 0,C 180,E1 19879.093,E2 19879.093} C_VEL
LIN {X 0,Y 402.688,Z 750.412,A -85,B 0,C 180,E1 19876.356,E2 19876.356} C_VEL
LIN {X 0,Y 404.211,Z 739.589,A -85,B 0,C 180,E1 19873.621,E2 19873.621} C_VEL
LIN {X 0,Y 406.112,Z 727.17,A -85,B 0,C 180,E1 19871.035,E2 19871.035} C_VEL
LIN {X 0,Y 408.37,Z 713.118,A -85,B 0,C 180,E1 19868.604,E2 19868.604} C_VEL
LIN {X 0,Y 410.813,Z 697.986,A -85,B 0,C 180,E1 19866.415,E2 19866.415} C_VEL
LIN {X 0,Y 413.351,Z 681.829,A -85,B 0,C 180,E1 19864.457,E2 19864.457} C_VEL
LIN {X 0,Y 415.977,Z 664.115,A -85,B 0,C 180,E1 19862.671,E2 19862.671} C_VEL
LIN {X 0,Y 418.461,Z 645.681,A -85,B 0,C 180,E1 19861.141,E2 19861.141} C_VEL
LIN {X 0,Y 420.773,Z 626.14,A -85,B 0,C 180,E1 19859.829,E2 19859.829} C_VEL
LIN {X 0,Y 422.718,Z 605.931,A -85,B 0,C 180,E1 19858.762,E2 19858.762} C_VEL
LIN {X 0,Y 424.307,Z 584.885,A -85,B 0,C 180,E1 19857.936,E2 19857.936} C_VEL
LIN {X 0,Y 426.886,Z 541.862,A -85,B 0,C 180,E1 19856.79,E2 19856.79} C_VEL
LIN {X 0,Y 431.575,Z 462.448,A -85,B 0,C 180,E1 19854.941,E2 19854.941} C_VEL
LIN {X 0,Y 434.785,Z 392.795,A -85,B 0,C 180,E1 19853.536,E2 19853.536} C_VEL
LIN {X 0,Y 436.618,Z 338.897,A -85,B 0,C 180,E1 19852.555,E2 19852.555} C_VEL
LIN {X 0,Y 437.224,Z 336.474,A -85,B 0,C 180,E1 19852.368,E2 19852.368} C_VEL
LIN {X 0,Y 437.422,Z 334.535,A -85,B 0,C 180,E1 19852.173,E2 19852.173} C_VEL
LIN {X 0,Y 430.069,Z 317.497,A -85,B 0,C 180,E1 19848.857,E2 19848.857} C_VEL
LIN {X 0,Y 423.985,Z 304.56,A -85,B 0,C 180,E1 19845.995,E2 19845.995} C_VEL
LIN {X 0,Y 417.976,Z 292.409,A -85,B 0,C 180,E1 19842.982,E2 19842.982} C_VEL
LIN {X 0,Y 412.809,Z 282.853,A -85,B 0,C 180,E1 19840.274,E2 19840.274} C_VEL
LIN {X 0,Y 410.141,Z 278.071,A -85,B 0,C 180,E1 19838.795,E2 19838.795} C_VEL
LIN {X 0,Y 408.062,Z 274.431,A -85,B 0,C 180,E1 19837.599,E2 19837.599} C_VEL
LIN {X 0,Y 407.326,Z 273.063,A -85,B 0,C 180,E1 19837.147,E2 19837.147} C_VEL
LIN {X 0,Y 405.244,Z 269.921,A -85,B 0,C 180,E1 19835.961,E2 19835.961} C_VEL
LIN {X 0,Y 404.873,Z 269.33,A -85,B 0,C 180,E1 19835.737,E2 19835.737} C_VEL
LIN {X 0,Y 403.754,Z 269.212,A -85,B 0,C 180,E1 19835.365,E2 19835.365} C_VEL
LIN {X 0,Y 411.531,Z 291.568,A -85,B 0,C 180,E1 19832.642,E2 19832.642} C_VEL
LIN {X 0,Y 414.831,Z 302.532,A -85,B 0,C 180,E1 19831.375,E2 19831.375} C_VEL
LIN {X 0,Y 413.47,Z 343.114,A -85,B 0,C 180,E1 19827.74,E2 19827.74} C_VEL
LIN {X 0,Y 411.892,Z 386.578,A -85,B 0,C 180,E1 19823.87,E2 19823.87} C_VEL
LIN {X 0,Y 410.246,Z 430.789,A -85,B 0,C 180,E1 19819.951,E2 19819.951} C_VEL
LIN {X 0,Y 409.368,Z 456.644,A -85,B 0,C 180,E1 19817.695,E2 19817.695} C_VEL
LIN {X 0,Y 406.614,Z 600.112,A -85,B 0,C 180,E1 19814.713,E2 19814.713} C_VEL
LIN {X 0,Y 406.38,Z 617.45,A -85,B 0,C 180,E1 19814.098,E2 19814.098} C_VEL
LIN {X 0,Y 405.934,Z 633.738,A -85,B 0,C 180,E1 19813.243,E2 19813.243} C_VEL
LIN {X 0,Y 405.366,Z 648.948,A -85,B 0,C 180,E1 19812.175,E2 19812.175} C_VEL
LIN {X 0,Y 404.693,Z 663.814,A -85,B 0,C 180,E1 19810.823,E2 19810.823} C_VEL
LIN {X 0,Y 404.007,Z 676.775,A -85,B 0,C 180,E1 19809.33,E2 19809.33} C_VEL
LIN {X 0,Y 403.369,Z 688.287,A -85,B 0,C 180,E1 19807.693,E2 19807.693} C_VEL
LIN {X 0,Y 402.786,Z 698.65,A -85,B 0,C 180,E1 19805.842,E2 19805.842} C_VEL
LIN {X 0,Y 402.372,Z 706.972,A -85,B 0,C 180,E1 19803.99,E2 19803.99} C_VEL
LIN {X 0,Y 402.047,Z 714.346,A -85,B 0,C 180,E1 19801.853,E2 19801.853} C_VEL
LIN {X 0,Y 401.87,Z 719.756,A -85,B 0,C 180,E1 19799.715,E2 19799.715} C_VEL
LIN {X 0,Y 401.814,Z 723.571,A -85,B 0,C 180,E1 19797.433,E2 19797.433} C_VEL
LIN {X 0,Y 401.874,Z 725.349,A -85,B 0,C 180,E1 19795.291,E2 19795.291} C_VEL
LIN {X 0,Y 402.029,Z 725.486,A -85,B 0,C 180,E1 19793.144,E2 19793.144} C_VEL
LIN {X 0,Y 402.281,Z 723.871,A -85,B 0,C 180,E1 19790.992,E2 19790.992} C_VEL
LIN {X 0,Y 402.691,Z 720.318,A -85,B 0,C 180,E1 19788.746,E2 19788.746} C_VEL
LIN {X 0,Y 403.162,Z 715.082,A -85,B 0,C 180,E1 19786.666,E2 19786.666} C_VEL
LIN {X 0,Y 403.79,Z 708.028,A -85,B 0,C 180,E1 19784.636,E2 19784.636} C_VEL
LIN {X 0,Y 404.5,Z 699.318,A -85,B 0,C 180,E1 19782.746,E2 19782.746} C_VEL
LIN {X 0,Y 405.231,Z 689.45,A -85,B 0,C 180,E1 19781.068,E2 19781.068} C_VEL
LIN {X 0,Y 406.002,Z 677.438,A -85,B 0,C 180,E1 19779.456,E2 19779.456} C_VEL
LIN {X 0,Y 406.695,Z 664.161,A -85,B 0,C 180,E1 19778.057,E2 19778.057} C_VEL
LIN {X 0,Y 407.227,Z 650.422,A -85,B 0,C 180,E1 19776.923,E2 19776.923} C_VEL
LIN {X 0,Y 407.626,Z 634.52,A -85,B 0,C 180,E1 19775.934,E2 19775.934} C_VEL
LIN {X 0,Y 407.813,Z 617.532,A -85,B 0,C 180,E1 19775.188,E2 19775.188} C_VEL
LIN {X 0,Y 407.753,Z 598.958,A -85,B 0,C 180,E1 19774.681,E2 19774.681} C_VEL
LIN {X 0,Y 409.494,Z 528.782,A -85,B 0,C 180,E1 19773.088,E2 19773.088} C_VEL
LIN {X 0,Y 411.613,Z 473.429,A -85,B 0,C 180,E1 19771.727,E2 19771.727} C_VEL
LIN {X 0,Y 414.066,Z 461.154,A -85,B 0,C 180,E1 19770.885,E2 19770.885} C_VEL
LIN {X 0,Y 415.505,Z 417.486,A -85,B 0,C 180,E1 19767.219,E2 19767.219} C_VEL
LIN {X 0,Y 415.99,Z 403.221,A -85,B 0,C 180,E1 19766.026,E2 19766.026} C_VEL
LIN {X 0,Y 418.451,Z 403.319,A -85,B 0,C 180,E1 19765.674,E2 19765.674} C_VEL
LIN {X 0,Y 422.077,Z 401.573,A -85,B 0,C 180,E1 19765.352,E2 19765.352} C_VEL
LIN {X 0,Y 427.082,Z 400.02,A -85,B 0,C 180,E1 19764.836,E2 19764.836} C_VEL
LIN {X 0,Y 429.69,Z 399.029,A -85,B 0,C 180,E1 19764.592,E2 19764.592} C_VEL
LIN {X 0,Y 439.403,Z 395.767,A -85,B 0,C 180,E1 19763.673,E2 19763.673} C_VEL
LIN {X 0,Y 442.192,Z 413.802,A -85,B 0,C 180,E1 19761.717,E2 19761.717} C_VEL
LIN {X 0,Y 446.536,Z 428.913,A -85,B 0,C 180,E1 19759.928,E2 19759.928} C_VEL
LIN {X 0,Y 453.049,Z 443.448,A -85,B 0,C 180,E1 19758.052,E2 19758.052} C_VEL
LIN {X 0,Y 460.716,Z 455.54,A -85,B 0,C 180,E1 19756.36,E2 19756.36} C_VEL
LIN {X 0,Y 470.56,Z 467.041,A -85,B 0,C 180,E1 19754.618,E2 19754.618} C_VEL
LIN {X 0,Y 471.953,Z 468.684,A -85,B 0,C 180,E1 19754.378,E2 19754.378} C_VEL
LIN {X 0,Y 461.259,Z 487.545,A -85,B 0,C 180,E1 19753.834,E2 19753.834} C_VEL
LIN {X 0,Y 451.391,Z 507.582,A -85,B 0,C 180,E1 19753.106,E2 19753.106} C_VEL
LIN {X 0,Y 442.924,Z 524.849,A -85,B 0,C 180,E1 19752.452,E2 19752.452} C_VEL
LIN {X 0,Y 436.8,Z 540.431,A -85,B 0,C 180,E1 19751.763,E2 19751.763} C_VEL
LIN {X 0,Y 434.453,Z 558.182,A -85,B 0,C 180,E1 19751.633,E2 19751.633} C_VEL
LIN {X 0,Y 433.185,Z 575.501,A -85,B 0,C 180,E1 19751.396,E2 19751.396} C_VEL
LIN {X 0,Y 431.684,Z 602.015,A -85,B 0,C 180,E1 19750.786,E2 19750.786} C_VEL
LIN {X 0,Y 429.239,Z 628.171,A -85,B 0,C 180,E1 19749.958,E2 19749.958} C_VEL
LIN {X 0,Y 426.798,Z 651.353,A -85,B 0,C 180,E1 19748.978,E2 19748.978} C_VEL
LIN {X 0,Y 424.009,Z 674.703,A -85,B 0,C 180,E1 19747.729,E2 19747.729} C_VEL
LIN {X 0,Y 421.107,Z 697.12,A -85,B 0,C 180,E1 19746.244,E2 19746.244} C_VEL
LIN {X 0,Y 418.088,Z 718.581,A -85,B 0,C 180,E1 19744.527,E2 19744.527} C_VEL
LIN {X 0,Y 415.287,Z 737.557,A -85,B 0,C 180,E1 19742.716,E2 19742.716} C_VEL
LIN {X 0,Y 412.347,Z 755.83,A -85,B 0,C 180,E1 19740.611,E2 19740.611} C_VEL
LIN {X 0,Y 409.767,Z 771.251,A -85,B 0,C 180,E1 19738.492,E2 19738.492} C_VEL
LIN {X 0,Y 407.192,Z 786.499,A -85,B 0,C 180,E1 19736.012,E2 19736.012} C_VEL
LIN {X 0,Y 405,Z 799.788,A -85,B 0,C 180,E1 19733.421,E2 19733.421} C_VEL
LIN {X 0,Y 403.18,Z 811.869,A -85,B 0,C 180,E1 19730.619,E2 19730.619} C_VEL
LIN {X 0,Y 401.741,Z 822.935,A -85,B 0,C 180,E1 19727.527,E2 19727.527} C_VEL
LIN {X 0,Y 400.785,Z 832.248,A -85,B 0,C 180,E1 19724.299,E2 19724.299} C_VEL
LIN {X 0,Y 400.282,Z 839.223,A -85,B 0,C 180,E1 19721.235,E2 19721.235} C_VEL
LIN {X 0,Y 400.063,Z 844.477,A -85,B 0,C 180,E1 19718.19,E2 19718.19} C_VEL
LIN {X 0,Y 399.998,Z 848.137,A -85,B 0,C 180,E1 19715.019,E2 19715.019} C_VEL
LIN {X 0,Y 399.997,Z 849.942,A -85,B 0,C 180,E1 19712.149,E2 19712.149} C_VEL
LIN {X 0,Y 400,Z 850.27,A -85,B 0,C 180,E1 19709.141,E2 19709.141} C_VEL
LIN {X 0,Y 399.99,Z 849.119,A -85,B 0,C 180,E1 19706.273,E2 19706.273} C_VEL
LIN {X 0,Y 400.017,Z 846.326,A -85,B 0,C 180,E1 19703.253,E2 19703.253} C_VEL
LIN {X 0,Y 400.145,Z 842.146,A -85,B 0,C 180,E1 19700.362,E2 19700.362} C_VEL
LIN {X 0,Y 400.503,Z 835.754,A -85,B 0,C 180,E1 19697.162,E2 19697.162} C_VEL
LIN {X 0,Y 401.199,Z 827.773,A -85,B 0,C 180,E1 19694.089,E2 19694.089} C_VEL
LIN {X 0,Y 402.278,Z 818.362,A -85,B 0,C 180,E1 19691.148,E2 19691.148} C_VEL
LIN {X 0,Y 403.889,Z 806.837,A -85,B 0,C 180,E1 19688.177,E2 19688.177} C_VEL
LIN {X 0,Y 405.925,Z 793.874,A -85,B 0,C 180,E1 19685.4,E2 19685.4} C_VEL
LIN {X 0,Y 408.25,Z 780.009,A -85,B 0,C 180,E1 19682.9,E2 19682.9} C_VEL
LIN {X 0,Y 411.049,Z 763.535,A -85,B 0,C 180,E1 19680.41,E2 19680.41} C_VEL
LIN {X 0,Y 413.893,Z 746.384,A -85,B 0,C 180,E1 19678.248,E2 19678.248} C_VEL
LIN {X 0,Y 416.702,Z 728.581,A -85,B 0,C 180,E1 19676.367,E2 19676.367} C_VEL
LIN {X 0,Y 419.587,Z 708.778,A -85,B 0,C 180,E1 19674.615,E2 19674.615} C_VEL
LIN {X 0,Y 422.649,Z 686.804,A -85,B 0,C 180,E1 19672.99,E2 19672.99} C_VEL
LIN {X 0,Y 425.4,Z 665.744,A -85,B 0,C 180,E1 19671.697,E2 19671.697} C_VEL
LIN {X 0,Y 428.247,Z 641.295,A -85,B 0,C 180,E1 19670.489,E2 19670.489} C_VEL
LIN {X 0,Y 430.84,Z 616.99,A -85,B 0,C 180,E1 19669.567,E2 19669.567} C_VEL
LIN {X 0,Y 432.997,Z 590.637,A -85,B 0,C 180,E1 19668.835,E2 19668.835} C_VEL
LIN {X 0,Y 434.363,Z 566.734,A -85,B 0,C 180,E1 19668.362,E2 19668.362} C_VEL
LIN {X 0,Y 437.078,Z 545.247,A -85,B 0,C 180,E1 19668.203,E2 19668.203} C_VEL
LIN {X 0,Y 438.231,Z 539.45,A -85,B 0,C 180,E1 19668.18,E2 19668.18} C_VEL
LIN {X 0,Y 446.859,Z 522.391,A -85,B 0,C 180,E1 19667.314,E2 19667.314} C_VEL
LIN {X 0,Y 456.833,Z 506.295,A -85,B 0,C 180,E1 19666.673,E2 19666.673} C_VEL
LIN {X 0,Y 462.365,Z 497.081,A -85,B 0,C 180,E1 19666.303,E2 19666.303} C_VEL
LIN {X 0,Y 452.76,Z 485.599,A -85,B 0,C 180,E1 19664.431,E2 19664.431} C_VEL
LIN {X 0,Y 445.671,Z 473.901,A -85,B 0,C 180,E1 19662.651,E2 19662.651} C_VEL
LIN {X 0,Y 439.804,Z 459.714,A -85,B 0,C 180,E1 19660.642,E2 19660.642} C_VEL
LIN {X 0,Y 436.212,Z 445.144,A -85,B 0,C 180,E1 19658.737,E2 19658.737} C_VEL
LIN {X 0,Y 434.345,Z 428.097,A -85,B 0,C 180,E1 19656.681,E2 19656.681} C_VEL
LIN {X 0,Y 434.571,Z 409.457,A -85,B 0,C 180,E1 19654.631,E2 19654.631} C_VEL
LIN {X 0,Y 437.552,Z 384.634,A -85,B 0,C 180,E1 19652.17,E2 19652.17} C_VEL
LIN {X 0,Y 441.281,Z 360.856,A -85,B 0,C 180,E1 19649.861,E2 19649.861} C_VEL
LIN {X 0,Y 430.073,Z 365.488,A -85,B 0,C 180,E1 19648.614,E2 19648.614} C_VEL
LIN {X 0,Y 424.378,Z 367.963,A -85,B 0,C 180,E1 19647.96,E2 19647.96} C_VEL
LIN {X 0,Y 420.372,Z 369.684,A -85,B 0,C 180,E1 19647.479,E2 19647.479} C_VEL
LIN {X 0,Y 418.715,Z 370.491,A -85,B 0,C 180,E1 19647.289,E2 19647.289} C_VEL
LIN {X 0,Y 415.423,Z 372.082,A -85,B 0,C 180,E1 19646.903,E2 19646.903} C_VEL
LIN {X 0,Y 413.863,Z 372.188,A -85,B 0,C 180,E1 19646.605,E2 19646.605} C_VEL
LIN {X 0,Y 412.808,Z 419.274,A -85,B 0,C 180,E1 19643.015,E2 19643.015} C_VEL
LIN {X 0,Y 411.457,Z 467.909,A -85,B 0,C 180,E1 19639.224,E2 19639.224} C_VEL
LIN {X 0,Y 410.178,Z 506.871,A -85,B 0,C 180,E1 19636.134,E2 19636.134} C_VEL
LIN {X 0,Y 408.299,Z 518.14,A -85,B 0,C 180,E1 19635.385,E2 19635.385} C_VEL
LIN {X 0,Y 406.118,Z 614.191,A -85,B 0,C 180,E1 19633.27,E2 19633.27} C_VEL
LIN {X 0,Y 406.208,Z 633.568,A -85,B 0,C 180,E1 19632.771,E2 19632.771} C_VEL
LIN {X 0,Y 406.144,Z 647.943,A -85,B 0,C 180,E1 19632.15,E2 19632.15} C_VEL
LIN {X 0,Y 405.857,Z 661.762,A -85,B 0,C 180,E1 19631.294,E2 19631.294} C_VEL
LIN {X 0,Y 405.411,Z 675.23,A -85,B 0,C 180,E1 19630.156,E2 19630.156} C_VEL
LIN {X 0,Y 404.841,Z 687.33,A -85,B 0,C 180,E1 19628.808,E2 19628.808} C_VEL
LIN {X 0,Y 404.203,Z 698.083,A -85,B 0,C 180,E1 19627.247,E2 19627.247} C_VEL
LIN {X 0,Y 403.584,Z 707.095,A -85,B 0,C 180,E1 19625.544,E2 19625.544} C_VEL
LIN {X 0,Y 403.057,Z 713.965,A -85,B 0,C 180,E1 19623.84,E2 19623.84} C_VEL
LIN {X 0,Y 402.605,Z 719.46,A -85,B 0,C 180,E1 19621.992,E2 19621.992} C_VEL
LIN {X 0,Y 402.217,Z 723.587,A -85,B 0,C 180,E1 19619.857,E2 19619.857} C_VEL
LIN {X 0,Y 401.967,Z 725.597,A -85,B 0,C 180,E1 19617.719,E2 19617.719} C_VEL
LIN {X 0,Y 401.828,Z 725.66,A -85,B 0,C 180,E1 19615.718,E2 19615.718} C_VEL
LIN {X 0,Y 401.793,Z 724.016,A -85,B 0,C 180,E1 19613.713,E2 19613.713} C_VEL
LIN {X 0,Y 401.857,Z 720.594,A -85,B 0,C 180,E1 19611.702,E2 19611.702} C_VEL
LIN {X 0,Y 402.046,Z 715.227,A -85,B 0,C 180,E1 19609.685,E2 19609.685} C_VEL
LIN {X 0,Y 402.344,Z 708.277,A -85,B 0,C 180,E1 19607.805,E2 19607.805} C_VEL
LIN {X 0,Y 402.756,Z 699.845,A -85,B 0,C 180,E1 19606.065,E2 19606.065} C_VEL
LIN {X 0,Y 403.253,Z 689.427,A -85,B 0,C 180,E1 19604.393,E2 19604.393} C_VEL
LIN {X 0,Y 403.788,Z 677.543,A -85,B 0,C 180,E1 19602.906,E2 19602.906} C_VEL
LIN {X 0,Y 404.291,Z 664.267,A -85,B 0,C 180,E1 19601.619,E2 19601.619} C_VEL
LIN {X 0,Y 404.722,Z 650.249,A -85,B 0,C 180,E1 19600.592,E2 19600.592} C_VEL
LIN {X 0,Y 405.002,Z 634.685,A -85,B 0,C 180,E1 19599.774,E2 19599.774} C_VEL
LIN {X 0,Y 405.099,Z 618.579,A -85,B 0,C 180,E1 19599.237,E2 19599.237} C_VEL
LIN {X 0,Y 406.893,Z 505.883,A -85,B 0,C 180,E1 19596.924,E2 19596.924} C_VEL
LIN {X 0,Y 407.559,Z 497.832,A -85,B 0,C 180,E1 19596.275,E2 19596.275} C_VEL
LIN {X 0,Y 409.24,Z 448.223,A -85,B 0,C 180,E1 19592.182,E2 19592.182} C_VEL
LIN {X 0,Y 410.905,Z 401.256,A -85,B 0,C 180,E1 19588.291,E2 19588.291} C_VEL
LIN {X 0,Y 412.534,Z 356.056,A -85,B 0,C 180,E1 19584.525,E2 19584.525} C_VEL
LIN {X 0,Y 413.649,Z 323.699,A -85,B 0,C 180,E1 19581.815,E2 19581.815} C_VEL
LIN {X 0,Y 415.297,Z 323.535,A -85,B 0,C 180,E1 19581.423,E2 19581.423} C_VEL
LIN {X 0,Y 418.093,Z 322.026,A -85,B 0,C 180,E1 19581.008,E2 19581.008} C_VEL
LIN {X 0,Y 419.381,Z 321.353,A -85,B 0,C 180,E1 19580.817,E2 19580.817} C_VEL
LIN {X 0,Y 422.565,Z 320.009,A -85,B 0,C 180,E1 19580.292,E2 19580.292} C_VEL
LIN {X 0,Y 424.667,Z 318.86,A -85,B 0,C 180,E1 19580.001,E2 19580.001} C_VEL
LIN {X 0,Y 429.522,Z 316.652,A -85,B 0,C 180,E1 19579.278,E2 19579.278} C_VEL
LIN {X 0,Y 434.472,Z 328.295,A -85,B 0,C 180,E1 19576.271,E2 19576.271} C_VEL
LIN {X 0,Y 438.36,Z 338.303,A -85,B 0,C 180,E1 19573.975,E2 19573.975} C_VEL
LIN {X 0,Y 437.876,Z 342.25,A -85,B 0,C 180,E1 19573.544,E2 19573.544} C_VEL
LIN {X 0,Y 437.65,Z 354.824,A -85,B 0,C 180,E1 19573.294,E2 19573.294} C_VEL
LIN {X 0,Y 434.969,Z 424.519,A -85,B 0,C 180,E1 19571.987,E2 19571.987} C_VEL
LIN {X 0,Y 430.958,Z 497.16,A -85,B 0,C 180,E1 19570.41,E2 19570.41} C_VEL
LIN {X 0,Y 429.211,Z 524.812,A -85,B 0,C 180,E1 19569.751,E2 19569.751} C_VEL
LIN {X 0,Y 427.948,Z 532.435,A -85,B 0,C 180,E1 19569.65,E2 19569.65} C_VEL
LIN {X 0,Y 421.711,Z 552.747,A -85,B 0,C 180,E1 19569.675,E2 19569.675} C_VEL
LIN {X 0,Y 420.657,Z 559.279,A -85,B 0,C 180,E1 19569.571,E2 19569.571} C_VEL
LIN {X 0,Y 418.686,Z 589.198,A -85,B 0,C 180,E1 19568.698,E2 19568.698} C_VEL
LIN {X 0,Y 416.997,Z 609.128,A -85,B 0,C 180,E1 19567.867,E2 19567.867} C_VEL
LIN {X 0,Y 414.883,Z 628.713,A -85,B 0,C 180,E1 19566.79,E2 19566.79} C_VEL
LIN {X 0,Y 412.337,Z 648.155,A -85,B 0,C 180,E1 19565.436,E2 19565.436} C_VEL
LIN {X 0,Y 409.711,Z 665.766,A -85,B 0,C 180,E1 19563.927,E2 19563.927} C_VEL
LIN {X 0,Y 406.777,Z 683.651,A -85,B 0,C 180,E1 19562.069,E2 19562.069} C_VEL
LIN {X 0,Y 403.908,Z 700.105,A -85,B 0,C 180,E1 19560.003,E2 19560.003} C_VEL
LIN {X 0,Y 401.244,Z 714.964,A -85,B 0,C 180,E1 19557.774,E2 19557.774} C_VEL
LIN {X 0,Y 398.862,Z 728.337,A -85,B 0,C 180,E1 19555.383,E2 19555.383} C_VEL
LIN {X 0,Y 396.709,Z 740.892,A -85,B 0,C 180,E1 19552.682,E2 19552.682} C_VEL
LIN {X 0,Y 395.082,Z 751.273,A -85,B 0,C 180,E1 19549.978,E2 19549.978} C_VEL
LIN {X 0,Y 393.856,Z 760.157,A -85,B 0,C 180,E1 19547.127,E2 19547.127} C_VEL
LIN {X 0,Y 393.016,Z 767.496,A -85,B 0,C 180,E1 19544.137,E2 19544.137} C_VEL
LIN {X 0,Y 392.551,Z 772.947,A -85,B 0,C 180,E1 19541.162,E2 19541.162} C_VEL
LIN {X 0,Y 392.324,Z 776.495,A -85,B 0,C 180,E1 19538.353,E2 19538.353} C_VEL
LIN {X 0,Y 392.221,Z 778.628,A -85,B 0,C 180,E1 19535.412,E2 19535.412} C_VEL
LIN {X 0,Y 392.193,Z 779.154,A -85,B 0,C 180,E1 19532.484,E2 19532.484} C_VEL
LIN {X 0,Y 392.238,Z 778.194,A -85,B 0,C 180,E1 19529.708,E2 19529.708} C_VEL
LIN {X 0,Y 392.353,Z 775.568,A -85,B 0,C 180,E1 19526.786,E2 19526.786} C_VEL
LIN {X 0,Y 392.635,Z 771.279,A -85,B 0,C 180,E1 19523.86,E2 19523.86} C_VEL
LIN {X 0,Y 393.133,Z 765.603,A -85,B 0,C 180,E1 19521.075,E2 19521.075} C_VEL
LIN {X 0,Y 394.024,Z 757.831,A -85,B 0,C 180,E1 19518.139,E2 19518.139} C_VEL
LIN {X 0,Y 395.29,Z 748.55,A -85,B 0,C 180,E1 19515.348,E2 19515.348} C_VEL
LIN {X 0,Y 397.04,Z 737.167,A -85,B 0,C 180,E1 19512.562,E2 19512.562} C_VEL
LIN {X 0,Y 399.07,Z 724.913,A -85,B 0,C 180,E1 19510.078,E2 19510.078} C_VEL
LIN {X 0,Y 401.403,Z 711.229,A -85,B 0,C 180,E1 19507.752,E2 19507.752} C_VEL
LIN {X 0,Y 403.987,Z 696.052,A -85,B 0,C 180,E1 19505.586,E2 19505.586} C_VEL
LIN {X 0,Y 406.655,Z 679.893,A -85,B 0,C 180,E1 19503.653,E2 19503.653} C_VEL
LIN {X 0,Y 409.273,Z 662.825,A -85,B 0,C 180,E1 19501.947,E2 19501.947} C_VEL
LIN {X 0,Y 411.789,Z 644.936,A -85,B 0,C 180,E1 19500.468,E2 19500.468} C_VEL
LIN {X 0,Y 414.087,Z 626.233,A -85,B 0,C 180,E1 19499.209,E2 19499.209} C_VEL
LIN {X 0,Y 416.073,Z 606.423,A -85,B 0,C 180,E1 19498.154,E2 19498.154} C_VEL
LIN {X 0,Y 417.692,Z 585.917,A -85,B 0,C 180,E1 19497.338,E2 19497.338} C_VEL
LIN {X 0,Y 420.545,Z 541.323,A -85,B 0,C 180,E1 19496.12,E2 19496.12} C_VEL
LIN {X 0,Y 425.34,Z 464.371,A -85,B 0,C 180,E1 19494.293,E2 19494.293} C_VEL
LIN {X 0,Y 428.647,Z 396.461,A -85,B 0,C 180,E1 19492.899,E2 19492.899} C_VEL
LIN {X 0,Y 430.711,Z 340.977,A -85,B 0,C 180,E1 19491.866,E2 19491.866} C_VEL
LIN {X 0,Y 431.307,Z 338.73,A -85,B 0,C 180,E1 19491.695,E2 19491.695} C_VEL
LIN {X 0,Y 424.458,Z 322.639,A -85,B 0,C 180,E1 19488.512,E2 19488.512} C_VEL
LIN {X 0,Y 418.319,Z 309.511,A -85,B 0,C 180,E1 19485.547,E2 19485.547} C_VEL
LIN {X 0,Y 412.817,Z 298.238,A -85,B 0,C 180,E1 19482.702,E2 19482.702} C_VEL
LIN {X 0,Y 407.753,Z 288.789,A -85,B 0,C 180,E1 19479.976,E2 19479.976} C_VEL
LIN {X 0,Y 405.269,Z 284.243,A -85,B 0,C 180,E1 19478.547,E2 19478.547} C_VEL
LIN {X 0,Y 402.491,Z 279.286,A -85,B 0,C 180,E1 19476.878,E2 19476.878} C_VEL
LIN {X 0,Y 400.475,Z 276.505,A -85,B 0,C 180,E1 19475.749,E2 19475.749} C_VEL
LIN {X 0,Y 398.394,Z 276.882,A -85,B 0,C 180,E1 19475.169,E2 19475.169} C_VEL
LIN {X 0,Y 398.326,Z 277.02,A -85,B 0,C 180,E1 19475.084,E2 19475.084} C_VEL
LIN {X 0,Y 405.95,Z 299.477,A -85,B 0,C 180,E1 19472.348,E2 19472.348} C_VEL
LIN {X 0,Y 407.517,Z 305.346,A -85,B 0,C 180,E1 19471.673,E2 19471.673} C_VEL
LIN {X 0,Y 406.059,Z 346.301,A -85,B 0,C 180,E1 19467.975,E2 19467.975} C_VEL
LIN {X 0,Y 404.426,Z 388.606,A -85,B 0,C 180,E1 19464.177,E2 19464.177} C_VEL
LIN {X 0,Y 402.689,Z 433.266,A -85,B 0,C 180,E1 19460.188,E2 19460.188} C_VEL
LIN {X 0,Y 401.79,Z 457.757,A -85,B 0,C 180,E1 19458.047,E2 19458.047} C_VEL
LIN {X 0,Y 398.871,Z 601.066,A -85,B 0,C 180,E1 19454.982,E2 19454.982} C_VEL
LIN {X 0,Y 398.622,Z 618.767,A -85,B 0,C 180,E1 19454.342,E2 19454.342} C_VEL
LIN {X 0,Y 398.179,Z 634.437,A -85,B 0,C 180,E1 19453.506,E2 19453.506} C_VEL
LIN {X 0,Y 397.633,Z 648.922,A -85,B 0,C 180,E1 19452.489,E2 19452.489} C_VEL
LIN {X 0,Y 396.959,Z 663.333,A -85,B 0,C 180,E1 19451.184,E2 19451.184} C_VEL
LIN {X 0,Y 396.28,Z 676.181,A -85,B 0,C 180,E1 19449.733,E2 19449.733} C_VEL
LIN {X 0,Y 395.572,Z 688.507,A -85,B 0,C 180,E1 19447.992,E2 19447.992} C_VEL
LIN {X 0,Y 395,Z 698.431,A -85,B 0,C 180,E1 19446.249,E2 19446.249} C_VEL
LIN {X 0,Y 394.516,Z 707.682,A -85,B 0,C 180,E1 19444.215,E2 19444.215} C_VEL
LIN {X 0,Y 394.191,Z 714.819,A -85,B 0,C 180,E1 19442.181,E2 19442.181} C_VEL
LIN {X 0,Y 393.994,Z 720.552,A -85,B 0,C 180,E1 19440.001,E2 19440.001} C_VEL
LIN {X 0,Y 393.921,Z 724.59,A -85,B 0,C 180,E1 19437.673,E2 19437.673} C_VEL
LIN {X 0,Y 393.986,Z 726.662,A -85,B 0,C 180,E1 19435.488,E2 19435.488} C_VEL
LIN {X 0,Y 394.164,Z 726.964,A -85,B 0,C 180,E1 19433.153,E2 19433.153} C_VEL
LIN {X 0,Y 394.442,Z 725.469,A -85,B 0,C 180,E1 19430.958,E2 19430.958} C_VEL
LIN {X 0,Y 394.865,Z 722.158,A -85,B 0,C 180,E1 19428.757,E2 19428.757} C_VEL
LIN {X 0,Y 395.368,Z 717.303,A -85,B 0,C 180,E1 19426.696,E2 19426.696} C_VEL
LIN {X 0,Y 396.028,Z 710.474,A -85,B 0,C 180,E1 19424.628,E2 19424.628} C_VEL
LIN {X 0,Y 396.752,Z 702.349,A -85,B 0,C 180,E1 19422.771,E2 19422.771} C_VEL
LIN {X 0,Y 397.602,Z 691.991,A -85,B 0,C 180,E1 19420.919,E2 19420.919} C_VEL
LIN {X 0,Y 398.417,Z 680.2,A -85,B 0,C 180,E1 19419.278,E2 19419.278} C_VEL
LIN {X 0,Y 399.117,Z 667.986,A -85,B 0,C 180,E1 19417.928,E2 19417.928} C_VEL
